# B&R Automation Studio project AGV
Automation Studio 4.12.2.93; technology packages: exosTechnology 2.1.0, mapp 5.20.0, mappCockpit 5.20.0, mappControl 5.20.0, mappMotion 5.20.1, mappView 5.20.0, mappVision 5.20.0

## Configuration CP1586

### Task classes (Cpu.sw)
```
Cyclic#1:
  motorCtrl <- ros_topics_typ.motorCtrl.prg
Binaries: FWRules, TCData, udbdef, User, iomap, Role, arconfig, asfw, ashwac, sysconf, ashwd, target, components
Libraries: ExOS, ExDeploy, ExData, runtime, sys_lib, FileIO, AsIOTime, ArEventLog, AsTCP, ros_topics, ROS, operator, astime, AsIecCon, brsystem, MTTypes, standard
```

## Configuration Config1

CPU X90CP174.48-00, AutomationRuntime B4.91, Build 6.3.0, Safety 0.0, Vc V4.72.6

### Task classes (Cpu.sw)
```
Cyclic#1 (cycle 5000 us, tolerance 0 us):
  motorCtrl <- ros_topics_typ.motorCtrl.prg
  VisionMain <- Package.VisionMain.prg
  WaterTank_ <- (binary)
NcDataObjects: mcdrivelog
Binaries: udbdef, FWRules, TCData, arcoal, arflatprv, arsvcreg, mvLoader, visionUnit, mCoWebSc, iomap, ashwac, Role, sysconf, arconfig, asfw, User, ashwd, target, components, Settings, viApp, viComp, ViLine
Libraries: brsystem, MTTypes, sys_lib, runtime, ROS, standard, ExOS, ExDeploy, ExData, FileIO, AsIOTime, ArEventLog, AsTCP, ros_topics, astime, ViBase, AsZip, AsARCfg, powerlnk, AsEPL, AsIO, MTBasics, MTFilter, AsIecCon, AsIODiag, AsETH, AsBrWStr, AsHttp, AsMem, AsBrStr, CoTrace, McBase, brdkViBase, brdkViCal, brdkViGeom, brdkViImg, brdkViMapp, brdkViVF, brdkWS, MTLinAlg, brdkMU, brdkSTR, AsSem, mpbase, arssl
```

### Hardware
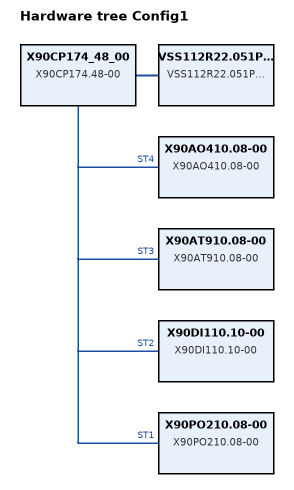
```
VSS112R22.051P-000 : VSS112R22.051P-000 v1.7.0.605  [PLK1 -> X90CP174_48_00.IF3 (NodeNumber=1) [Cable Type=PowerlinkCable, Length=10, Version=1.0.0.3]]
  Supervision = off
  VisionConfig = gCamera
X90AO410.08-00 : X90AO410.08-00 v1.1.0.0  [ST -> X90CP174_48_00.ST4]
X90AT910.08-00 : X90AT910.08-00 v1.0.1.0  [ST -> X90CP174_48_00.ST3]
X90CP174_48_00 : X90CP174.48-00 v1.4.5.0  [X1 -> X1.SL]
  Module X1 (Type=X1, Virtual=true, Version=1.4.5.0)
    Connection (Connector=SL, TargetModule=X90CP174_48_00, TargetConnector=X1)
    ChannelConfig01 = 42
    DigitalFilterPin01 = 0
    ChannelConfig02 = 42
    DigitalFilterPin02 = 0
    ChannelConfig03 = 42
    DigitalFilterPin03 = 0
    ChannelConfig04 = 42
    DigitalFilterPin04 = 0
    IN1_CounterFunction01 = 3
    IN1_CounterFunction02 = 3
    ChannelConfig33 = 15
    PWMSource33 = 1
    PWMSyncPeriod33 = 125
    ChannelConfig34 = 20
    ChannelConfig35 = 20
    ChannelConfig36 = 20  // Configuration and impedance of pin X1.A.J1  
    ChannelConfig37 = 16
    ChannelConfig38 = 20  // Configuration and impedance of pin X1.A.L1  (6A)
    ChannelConfig39 = 20  // Configuration and impedance of pin X1.A.M2 (6A)
    ChannelConfig40 = 20
    ChannelConfig41 = 15
    PWMSource41 = 1
    PWMSyncPeriod41 = 125
    PWMDisplacement41 = 62
    ChannelConfig42 = 20
    ChannelConfig43 = 20  // Configuration and impedance of pin X1.B.H1  (6A)
    ChannelConfig44 = 20  // Configuration and impedance of pin X1.B.H3  (6A)
    ChannelConfig45 = 16  // Configuration and impedance of pin X1.B.G4  (6A)
    ChannelConfig46 = 20
    ChannelConfig47 = 20
    ChannelConfig48 = 20
  Connector IF2:
    ActivateDevice = 1
    Mode = Manual
    InternetAddress = 192.168.87.200
    SubnetMask = 255.255.255.0
    InaNodeNumber = 1
  Connector IF3:
    MtuSize = 1500
    CycleTime = 5000
    InternetAddress = 192.168.200.240
    SubnetMask = 255.255.255.0
  ConfigurationID = AGV_Config1
  UserPartitionSize = 0
  EnableUsbRemoteInstall = 1
  EnableCfRemoteInstall = 1
  TimerDeviceType = EPLX2X
  TimerDevice = X90CP174_48_00.IF3
  TaskClassIdleTime = 5000
  Cyclic1Duration = 5000
  Cyclic1Tolerance = 0
  Cyclic1Stack = 16384
  Cyclic2Duration = 20000
  Cyclic2Tolerance = 20000
  Cyclic3Duration = 50000
  Cyclic3Tolerance = 50000
  Cyclic4Duration = 100000
  Cyclic4Tolerance = 100000
  Cyclic5Duration = 200000
  Cyclic5Tolerance = 200000
  Cyclic6Duration = 500000
  Cyclic6Tolerance = 500000
  Cyclic7Duration = 1000000
  Cyclic7Tolerance = 1000000
  Cyclic8Duration = 10000
  Cyclic8Tolerance = 30000000
  FileDevice1
  FileDeviceName1 = USER
  FileDevicePath1 = USER_PATH
  Route1
  DestinationAddress1 = 10.0.0.2
  SubnetMask1 = 255.255.255.0
  ActivateOpcUa = 1
  OpcUaInformationModels_PV_Version = 2
  OpcUaInformationModel_BaseObjectTypeForStructures = 0
X90DI110.10-00 : X90DI110.10-00 v1.1.1.0  [ST -> X90CP174_48_00.ST2]
X90PO210.08-00 : X90PO210.08-00 v1.4.0.0  [ST -> X90CP174_48_00.ST1]
```

### IoMap.iom - X90CP174_48_00/IoMap.iom
```iecst
VAR_CONFIG
	::motorCtrl:localVariables[0].hw.output.pwm AT %QW."X1".PWMOutput33;
	::motorCtrl:localVariables[0].hw.input.encoder AT %IW."X1".Encoder01;
	::motorCtrl:localVariables[0].hw.input.current[0] AT %IW."X1".Current33;
	::motorCtrl:localVariables[0].hw.input.current[1] AT %IW."X1".Current34;
	::motorCtrl:localVariables[0].hw.input.current[2] AT %IW."X1".Current35;
	::motorCtrl:localVariables[0].hw.input.current[3] AT %IW."X1".Current36;
	::motorCtrl:localVariables[0].hw.input.overload AT %IX."X1".OverloadDigitalOutput33;
	::motorCtrl:localVariables[0].hw.output.clear AT %QX."X1".OverloadClear33;
	::motorCtrl:localVariables[1].hw.input.encoder AT %IW."X1".Encoder02;
	::motorCtrl:localVariables[1].hw.output.pwm AT %QW."X1".PWMOutput37;
	::motorCtrl:localVariables[0].hw.input.current[4] AT %IW."X1".Current37;
	::motorCtrl:localVariables[0].hw.input.current[6] AT %IW."X1".Current39;
	::motorCtrl:localVariables[1].hw.input.nettime AT %ID."X90CP174_48_00".SystemTime;
	::motorCtrl:localVariables[0].hw.input.nettime AT %ID."X90CP174_48_00".SystemTime;
	::motorCtrl:localVariables[0].hw.input.current[5] AT %IW."X1".Current38;
	::motorCtrl:localVariables[0].hw.input.current[7] AT %IW."X1".Current40;
	::motorCtrl:localVariables[1].hw.output.pwm AT %QW."X1".PWMOutput41;
	::motorCtrl:localVariables[1].hw.output.clear AT %QX."X1".OverloadClear41;
	::motorCtrl:localVariables[1].hw.input.current[0] AT %IW."X1".Current41;
	::motorCtrl:localVariables[1].hw.input.overload AT %IX."X1".OverloadDigitalOutput41;
	::motorCtrl:localVariables[1].hw.input.current[1] AT %IW."X1".Current42;
	::motorCtrl:localVariables[1].hw.input.current[2] AT %IW."X1".Current43;
	::motorCtrl:localVariables[1].hw.input.current[3] AT %IW."X1".Current44;
	::motorCtrl:localVariables[1].hw.input.current[4] AT %IW."X1".Current45;
	::motorCtrl:localVariables[1].hw.input.current[5] AT %IW."X1".Current46;
	::motorCtrl:localVariables[1].hw.input.current[6] AT %IW."X1".Current47;
	::motorCtrl:localVariables[1].hw.input.current[7] AT %IW."X1".Current48;
	::VisionMain:hwCam.in.common.moduleOk AT %IX."VSS112R22.051P-000".ModuleOk;
	::VisionMain:hwCam.in.common.serialNumber AT %ID."VSS112R22.051P-000".SerialNumber;
	::VisionMain:hwCam.in.common.moduleId AT %ID."VSS112R22.051P-000".ModuleID;
	::VisionMain:hwCam.in.common.hardwareVariant AT %ID."VSS112R22.051P-000".HardwareVariant;
	::VisionMain:hwCam.in.common.firmwareVersion AT %ID."VSS112R22.051P-000".FirmwareVersion;
	::VisionMain:hwCam.in.status.sensorTemperature AT %IB."VSS112R22.051P-000".SensorTemperature;
	::VisionMain:hwCam.in.status.lightWarningCnt AT %IB."VSS112R22.051P-000".LightWarningCnt;
	::VisionMain:hwCam.out.par.statusLED AT %QB."VSS112R22.051P-000".StatusLED;
	::VisionMain:hwCam.in.status.cameraStatus AT %ID."VSS112R22.051P-000".CameraStatus;
	::VisionMain:hwCam.in.status.acceptedAcquisitionCnt AT %IB."VSS112R22.051P-000".AcceptedAcquisitionCnt;
	::VisionMain:hwCam.in.status.completedAcquisitionCnt AT %IB."VSS112R22.051P-000".CompletedAcquisitionCnt;
	::VisionMain:hwCam.in.status.failedAcquisitionCnt AT %IB."VSS112R22.051P-000".FailedAcquisitionCnt;
	::VisionMain:hwCam.in.status.gainLevel AT %IB."VSS112R22.051P-000".ReadGainLevel;
	::VisionMain:hwCam.in.status.focus AT %IW."VSS112R22.051P-000".ReadFocus;
	::VisionMain:hwCam.in.status.exposureTime AT %ID."VSS112R22.051P-000".ReadExposureTime;
	::VisionMain:hwCam.out.par.gainLevel AT %QB."VSS112R22.051P-000".GainLevel;
	::VisionMain:hwCam.out.par.focus AT %QW."VSS112R22.051P-000".SetFocus;
	::VisionMain:hwCam.out.par.exposureTime AT %QD."VSS112R22.051P-000".ExposureTime01;
	::VisionMain:hwCam.out.par.delayNetTime AT %QD."VSS112R22.051P-000".DelayNettime01;
	::VisionMain:hwCam.out.par.flashColor AT %QB."VSS112R22.051P-000".FlashColor01;
	::VisionMain:hwCam.out.par.flashSegment AT %QB."VSS112R22.051P-000".FlashSegment01;
	::VisionMain:hwCam.in.status.undervoltageError AT %IX."VSS112R22.051P-000".UndervoltageError;
	::VisionMain:hwCam.in.status.digitalInput AT %IX."VSS112R22.051P-000".DigitalInput01;
	::VisionMain:hwCam.out.cmd.digitalOutput AT %QX."VSS112R22.051P-000".DigitalOutput01;
	::VisionMain:hwCam.in.status.digitalOutputStatus AT %IX."VSS112R22.051P-000".DigitalOutputStatus01;
	::VisionMain:hwCam.in.status.imageAcquisitionReady AT %IX."VSS112R22.051P-000".ImageAcquisitionReady;
	::VisionMain:hwCam.in.status.imageProcessingActive AT %IX."VSS112R22.051P-000".ImageProcessingActive;
	::VisionMain:hwCam.out.cmd.imageAcquisition AT %QX."VSS112R22.051P-000".ImageAcquisition;
	::VisionMain:hwCam.out.cmd.resetAcquisiton AT %QX."VSS112R22.051P-000".ResetAcquisition;
	::VisionMain:hwCam.out.cmd.searchAcquisitonSettings AT %QX."VSS112R22.051P-000".SearchAcquisitionSettings;
	::VisionMain:hwCam.out.par.IRFilter AT %QX."VSS112R22.051P-000".IRFilter;
	::VisionMain:hwCam.out.par.chromaticLock AT %QX."VSS112R22.051P-000".ChromaticLock;
	::VisionMain:hwCam.in.status.cameraProcessingTime AT %IW."VSS112R22.051P-000".CameraProcessingTime;
	::VisionMain:hwCam.in.status.imageProcessingError AT %IW."VSS112R22.051P-000".ImageProcessingError;
	::VisionMain:hwCam.in.status.imageNettime AT %ID."VSS112R22.051P-000".ImageNettime;
	::VisionMain:hwBlob.out.common.enable AT %QX."VSS112R22.051P-000".Enable;
	::VisionMain:hwBlob.out.common.numSearchMax AT %QB."VSS112R22.051P-000".NumSearchMax;
	::VisionMain:hwBlob.out.regionFeatures AT %QX."VSS112R22.051P-000".RegionalFeatures;
	::VisionMain:hwBlob.out.enhancedBlobInformation AT %QX."VSS112R22.051P-000".EnhancedBlobInfo;
	::VisionMain:hwBlob.out.common.alignment AT %QB."VSS112R22.051P-000".Alignment;
	::VisionMain:hwBlob.out.common.offsetROI.x AT %QD."VSS112R22.051P-000".OffsetRoiX;
	::VisionMain:hwBlob.out.common.offsetROI.y AT %QD."VSS112R22.051P-000".OffsetRoiY;
	::VisionMain:hwBlob.out.common.offsetROI.orientation AT %QW."VSS112R22.051P-000".OffsetRoiOrientation;
	::VisionMain:hwBlob.out.common.offsetROI.rotCenterX AT %QD."VSS112R22.051P-000".OffsetRoiRotationCenterX;
	::VisionMain:hwBlob.out.common.offsetROI.rotCenterY AT %QD."VSS112R22.051P-000".OffsetRoiRotationCenterY;
	::VisionMain:hwBlob.in.results[0].xMin AT %ID."VSS112R22.051P-000".BlobXMin01;
	::VisionMain:hwBlob.in.results[0].xMax AT %ID."VSS112R22.051P-000".BlobXMax01;
	::VisionMain:hwBlob.in.results[0].yMin AT %ID."VSS112R22.051P-000".BlobYMin01;
	::VisionMain:hwBlob.in.results[0].yMax AT %ID."VSS112R22.051P-000".BlobYMax01;
	::VisionMain:hwBlob.in.common.numResults AT %IB."VSS112R22.051P-000".NumRes;
	::motorCtrl:suction.valveEnable AT %QX."X90PO210.08-00".DigitalOutput01;
	::motorCtrl:suction.motorEnable AT %QX."X90PO210.08-00".DigitalOutput02;
	::VisionMain:hwBlob.in.results[0].area AT %ID."VSS112R22.051P-000".blobArea01;
	::VisionMain:hwBlob.in.results[1].area AT %ID."VSS112R22.051P-000".blobArea02;
	::VisionMain:hwBlob.in.results[1].xMin AT %ID."VSS112R22.051P-000".BlobXMin02;
	::VisionMain:hwBlob.in.results[1].xMax AT %ID."VSS112R22.051P-000".BlobXMax02;
	::VisionMain:hwBlob.in.results[1].yMin AT %ID."VSS112R22.051P-000".BlobYMin02;
	::VisionMain:hwBlob.in.results[1].yMax AT %ID."VSS112R22.051P-000".BlobYMax02;
	::VisionMain:hwBlob.in.results[0].modelNumber AT %IB."VSS112R22.051P-000".model01;
	::VisionMain:hwBlob.in.results[1].modelNumber AT %IB."VSS112R22.051P-000".model02;
	::VisionMain:hwBlob.in.results[2].modelNumber AT %IB."VSS112R22.051P-000".model03;
	::VisionMain:hwBlob.in.results[3].modelNumber AT %IB."VSS112R22.051P-000".model04;
	::VisionMain:hwBlob.in.results[2].area AT %ID."VSS112R22.051P-000".blobArea03;
	::VisionMain:hwBlob.in.results[3].area AT %ID."VSS112R22.051P-000".blobArea04;
	::VisionMain:hwBlob.in.results[2].xMin AT %ID."VSS112R22.051P-000".BlobXMin03;
	::VisionMain:hwBlob.in.results[3].xMin AT %ID."VSS112R22.051P-000".BlobXMin04;
	::VisionMain:hwBlob.in.results[2].xMax AT %ID."VSS112R22.051P-000".BlobXMax03;
	::VisionMain:hwBlob.in.results[3].xMax AT %ID."VSS112R22.051P-000".BlobXMax04;
	::VisionMain:hwBlob.in.results[2].yMin AT %ID."VSS112R22.051P-000".BlobYMin03;
	::VisionMain:hwBlob.in.results[3].yMin AT %ID."VSS112R22.051P-000".BlobYMin04;
	::VisionMain:hwBlob.in.results[2].yMax AT %ID."VSS112R22.051P-000".BlobYMax03;
	::VisionMain:hwBlob.in.results[3].yMax AT %ID."VSS112R22.051P-000".BlobYMax04;
	::VisionMain:hwBlob.in.results[0].positionX AT %ID."VSS112R22.051P-000".posX01;
	::VisionMain:hwBlob.in.results[1].positionX AT %ID."VSS112R22.051P-000".posX02;
	::VisionMain:hwBlob.in.results[2].positionX AT %ID."VSS112R22.051P-000".posX03;
	::VisionMain:hwBlob.in.results[3].positionX AT %ID."VSS112R22.051P-000".posX04;
	::VisionMain:hwBlob.in.results[0].positionY AT %ID."VSS112R22.051P-000".posY01;
	::VisionMain:hwBlob.in.results[1].positionY AT %ID."VSS112R22.051P-000".posY02;
	::VisionMain:hwBlob.in.results[2].positionY AT %ID."VSS112R22.051P-000".posY03;
	::VisionMain:hwBlob.in.results[3].positionY AT %ID."VSS112R22.051P-000".posY04;
	::VisionMain:hwBlob.in.results[0].circularity AT %IB."VSS112R22.051P-000".blobCirc01;
	::VisionMain:hwBlob.in.results[1].circularity AT %IB."VSS112R22.051P-000".blobCirc02;
	::VisionMain:hwBlob.in.results[2].circularity AT %IB."VSS112R22.051P-000".blobCirc03;
	::VisionMain:hwBlob.in.results[3].circularity AT %IB."VSS112R22.051P-000".blobCirc04;
	::VisionMain:hwBlob.in.results[0].rectangularity AT %IB."VSS112R22.051P-000".blobRect01;
	::VisionMain:hwBlob.in.results[1].rectangularity  AT %IB."VSS112R22.051P-000".blobRect02;
	::VisionMain:hwBlob.in.results[2].rectangularity  AT %IB."VSS112R22.051P-000".blobRect03;
	::VisionMain:hwBlob.in.results[3].rectangularity  AT %IB."VSS112R22.051P-000".blobRect04;
END_VAR
```

### target.exostarget - X90CP174_48_00/exosTechnology/target.exostarget
```
Element gTarget_0 (Type=exostarget)
  General:
    ConnectionIP = 192.168.87.42
    Logging:
      LogLevel = Success
      LogFilters:
        LogFilterUser = On
        LogFilterSystem = On
        LogFilterVerbose = Off
      LogDestination = Volatile
    Deployment = On
      MaxRestarts = 10
    DataConnection = On
      ConnectionType = TCPIP
      TimeSynchronization:
        TimeConnection:
          TimePort = 49001
        PrecisionUsec = 5000
        GuardTimeSec = 180
        DeviationPerHourUsec = 100000
      DataConnectionLogging:
        LogConnection:
          LogPort = 49002
          LogShmPath = exos_log
        LogCycleTimeMsec = 50
  Components:
    ComponentsGeneral:
      ComponentsHeartbeatMsec = 500
      ComponentsTimeoutSec = 2
      ComponentsTaskClass = 2
      ComponentsCycleTimeMsec = 10
    Component[0]:
      ComponentConfigurationLink = gros_topics_typ_0
      DataModels:
        Instance[0]:
          InstanceName = ros_topics_typ_0
          InstanceConnection:
            InstancePort = 49005
            InstanceShmPath = ros_topics_typ_0
  ComponentDataConnection:
    Version = 2.1.0-1
    ErrorHandling = Target
    RestartEvent = Target
    StartupTimeout = 5
    Predefined:
      Files:
        File[0]:
          FileName = ufw-exos-data
          ChangeEvent = Ignore
        File[1]:
          FileName = exos-data-ufw-profile.sh
          ChangeEvent = Ignore
        File[2]:
          FileName = exos-data-ports-allow.sh
          ChangeEvent = Restart
        File[3]:
          FileName = exos-data.conf
          ChangeEvent = Restart
        File[4]:
          FileName = exos-data_2.1.0-1_amd64.deb
          ChangeEvent = Reinstall
        File[5]:
          FileName = exos-data-eth_2.1.0-1_amd64.deb
          ChangeEvent = Reinstall
        File[6]:
          FileName = exos-data-remove.sh
          ChangeEvent = Ignore
        File[7]:
          FileName = run_server.sh
          ChangeEvent = Ignore
        File[8]:
          FileName = setup_build_environment.sh
          ChangeEvent = Ignore
        File[9]:
          FileName = libzmq5_4.2.1-4+deb9u2_amd64.deb
          ChangeEvent = Reinstall
        File[10]:
          FileName = libpgm-5.2-0_5.2.122~dfsg-2_amd64.deb
          ChangeEvent = Reinstall
        File[11]:
          FileName = libsodium18_1.0.11-2_amd64.deb
          ChangeEvent = Reinstall
      Services:
        Service[0]:
          Type = Install
          Command = dpkg -i *.deb
          WorkingDirectory
        Service[1]:
          Type = Remove
          Command = dpkg --purge exos-data
          WorkingDirectory
        Service[2]:
          Type = Remove
          Command = dpkg --purge exos-data-eth
          WorkingDirectory
        Service[3]:
          Type = Remove
          Command = sh exos-data-remove.sh
          WorkingDirectory
        Service[4]:
          Type = Startup
          Command = cp exos-data.conf /etc/exos-data.conf
          WorkingDirectory
        Service[5]:
          Type = Startup
          Command = sh exos-data-ufw-profile.sh
          WorkingDirectory
        Service[6]:
          Type = Startup
          Command = sh exos-data-ports-allow.sh
          WorkingDirectory
        Service[7]:
          Type = Runtime
          Command = /usr/bin/exos_mr
          WorkingDirectory
  Simulation:
    SimConnectionIP = 192.168.87.42
    SimDeployment = On
    SimDataConnection = On
      SimConnectionType = TCPIP
      SimTimeSynchronization:
        SimPrecisionUsec = 10000
        SimGuardTimeSec = 30
    SimComponentsGeneral:
      SimComponentsHeartbeatMsec = 1000
      SimComponentsTimeoutSec = 75
```

### viComp.visioncomponent - X90CP174_48_00/mappVision/viComp.visioncomponent
```
Element gCamera (Type=visioncomponent)
  VisionApplicationReference = ViLine
```

## Logical view

Binary libraries used (declarations not repeated): operator, runtime, astime, AsIecCon, brsystem, standard, MTTypes, sys_lib, ROS, FileIO, AsIOTime, ArEventLog, AsTCP, ExOS, ExDeploy, ExData, AsZip, AsARCfg, powerlnk, AsEPL, AsIO, AsIODiag, AsETH, AsBrWStr, AsHttp, AsMem, AsBrStr, brdkViBase 1.00.4, brdkViCal, brdkViGeom, brdkViImg, brdkViMapp, brdkViVF, brdkWS, McBase 5.20.1, ViBase, CoTrace, MTBasics 5.20.0, MTFilter 5.20.0, MTLinAlg, brdkMU, brdkSTR, AsSem

### Global.var - Global variables
```iecst
VAR
	updateLineStatus : BOOL;
	sharpTurn : BOOL;
	rightTurn : BOOL;
	orientationReached : BOOL := TRUE;
	lineMode : BOOL;
	drejMere : REAL;
	Test2 : INT;
	slowDown : REAL;
	angVel : LREAL;
	holdRight : BOOL;
	lineFollow : ros_lineMode;
	moveForward : BOOL;
	lineStatus : ros_lineStatus;
	awaitDecision : BOOL;
	tempDec : BOOL;
	sammenEnable : BOOL;
END_VAR
```

### Package Logical/Libraries - Global libraries

- ros_topics_typ.exospkg (not shown)

### exos_ros_topics_typ.h - Generated datamodel header for ros_topics_typ
```c
/*Automatically generated header file from ros_topics_typ.typ*/

#ifndef _EXOS_COMP_ROS_TOPICS_TYP_H_
#define _EXOS_COMP_ROS_TOPICS_TYP_H_

#include "exos_api.h"

#if defined(_SG4)
#include <ros_topics.h>
#else
#include <stddef.h>
#include <stdint.h>
#include <stdbool.h>

typedef struct ros_lineStatus
{
    int16_t lineStatusCode;

} ros_lineStatus;

typedef struct ros_lineMode
{
    bool lineMode;
    bool lineSharpTurn;
    bool lineHoldRight;
    bool lineForward;
    bool lineInterSection;
    bool lineDecision;
    bool lineFast;
    bool lineSlow;

} ros_lineMode;

typedef struct ros_armBools
{
    bool vaccumValve;
    bool vaccumMotor;

} ros_armBools;

typedef struct ros_encoder
{
    int16_t encoder1;
    int16_t encoder2;

} ros_encoder;

typedef struct ros_config_typ
{
    double maxSpeed;
    double minSpeed;
    double baseWidth;

} ros_config_typ;

typedef struct ros_topic_vector3_typ
{
    double y;
    double z;
    double x;

} ros_topic_vector3_typ;

typedef struct ros_topic_twist_typ
{
    struct ros_topic_vector3_typ angular;
    struct ros_topic_vector3_typ linear;

} ros_topic_twist_typ;

typedef struct ros_topic_time_typ
{
    uint32_t nsec;
    uint32_t sec;

} ros_topic_time_typ;

typedef struct ros_topic_header_typ
{
    struct ros_topic_time_typ stamp;
    uint32_t seq;
    char frame_id[21];

} ros_topic_header_typ;

typedef struct ros_topic_twistCor_typ
{
    struct ros_topic_twist_typ twist;

} ros_topic_twistCor_typ;

typedef struct ros_topic_quaternion_typ
{
    double y;
    double z;
    double w;
    double x;

} ros_topic_quaternion_typ;

typedef struct ros_topic_point_typ
{
    double y;
    double z;
    double x;

} ros_topic_point_typ;

typedef struct ros_topic_pose_typ
{
    struct ros_topic_point_typ position;
    struct ros_topic_quaternion_typ orientation;

} ros_topic_pose_typ;

typedef struct ros_topic_poseCor_typ
{
    struct ros_topic_pose_typ pose;

} ros_topic_poseCor_typ;

typedef struct ros_topic_odemety_typ
{
    struct ros_topic_poseCor_typ pose;
    struct ros_topic_twistCor_typ twist;
    struct ros_topic_header_typ header;

} ros_topic_odemety_typ;

typedef struct ros_topics_typ
{
    struct ros_topic_odemety_typ odemetry; //PUB
    struct ros_topic_twist_typ twist; //SUB
    struct ros_config_typ config; //SUB
    struct ros_encoder encoder; //PUB
    struct ros_armBools vaccumTopic; //SUB
    struct ros_lineMode lineFollow; //SUB
    struct ros_lineStatus lineStatus; //PUB

} ros_topics_typ;

#endif // _SG4

EXOS_ERROR_CODE exos_datamodel_connect_ros_topics_typ(exos_datamodel_handle_t *datamodel, exos_datamodel_event_cb datamodel_event_callback);

#endif // _EXOS_COMP_ROS_TOPICS_TYP_H_
```

### libros_topics_typ.h - ros_topics_typ static library wrapper header
```c
#ifndef _LIBROS_TOPICS_TYP_H_
#define _LIBROS_TOPICS_TYP_H_

#include "exos_ros_topics_typ.h"

typedef void (*libros_topics_typ_event_cb)(void);
typedef void (*libros_topics_typ_method_fn)(void);
typedef int32_t (*libros_topics_typ_get_nettime_fn)(void);
typedef void (*libros_topics_typ_log_fn)(char *log_entry);

typedef struct libros_topics_typodemetry
{
    libros_topics_typ_event_cb on_change;
    int32_t nettime;
    ros_topic_odemety_typ value;
} libros_topics_typodemetry_t;

typedef struct libros_topics_typtwist
{
    libros_topics_typ_method_fn publish;
    ros_topic_twist_typ value;
} libros_topics_typtwist_t;

typedef struct libros_topics_typconfig
{
    libros_topics_typ_method_fn publish;
    ros_config_typ value;
} libros_topics_typconfig_t;

typedef struct libros_topics_typencoder
{
    libros_topics_typ_event_cb on_change;
    int32_t nettime;
    ros_encoder value;
} libros_topics_typencoder_t;

typedef struct libros_topics_typvaccumTopic
{
    libros_topics_typ_method_fn publish;
    ros_armBools value;
} libros_topics_typvaccumTopic_t;

typedef struct libros_topics_typlineFollow
{
    libros_topics_typ_method_fn publish;
    ros_lineMode value;
} libros_topics_typlineFollow_t;

typedef struct libros_topics_typlineStatus
{
    libros_topics_typ_event_cb on_change;
    int32_t nettime;
    ros_lineStatus value;
} libros_topics_typlineStatus_t;

typedef struct libros_topics_typ_log
{
    libros_topics_typ_log_fn error;
    libros_topics_typ_log_fn warning;
    libros_topics_typ_log_fn success;
    libros_topics_typ_log_fn info;
    libros_topics_typ_log_fn debug;
    libros_topics_typ_log_fn verbose;
} libros_topics_typ_log_t;

typedef struct libros_topics_typ
{
    libros_topics_typ_method_fn connect;
    libros_topics_typ_method_fn disconnect;
    libros_topics_typ_method_fn process;
    libros_topics_typ_method_fn set_operational;
    libros_topics_typ_method_fn dispose;
    libros_topics_typ_get_nettime_fn get_nettime;
    libros_topics_typ_log_t log;
    libros_topics_typ_event_cb on_connected;
    libros_topics_typ_event_cb on_disconnected;
    libros_topics_typ_event_cb on_operational;
    bool is_connected;
    bool is_operational;
    libros_topics_typodemetry_t odemetry;
    libros_topics_typtwist_t twist;
    libros_topics_typconfig_t config;
    libros_topics_typencoder_t encoder;
    libros_topics_typvaccumTopic_t vaccumTopic;
    libros_topics_typlineFollow_t lineFollow;
    libros_topics_typlineStatus_t lineStatus;
} libros_topics_typ_t;

#ifdef __cplusplus
extern "C" {
#endif
libros_topics_typ_t *libros_topics_typ_init(void);
#ifdef __cplusplus
}
#endif
#endif // _LIBROS_TOPICS_TYP_H_
```

### libros_topics_typ.c - ros_topics_typ static library wrapper source
```c
#include <string.h>
#define EXOS_ASSERT_LOG &logger
#include "exos_log.h"
#include "libros_topics_typ.h"

#define SUCCESS(_format_, ...) exos_log_success(&logger, EXOS_LOG_TYPE_USER, _format_, ##__VA_ARGS__);
#define INFO(_format_, ...) exos_log_info(&logger, EXOS_LOG_TYPE_USER, _format_, ##__VA_ARGS__);
#define VERBOSE(_format_, ...) exos_log_debug(&logger, EXOS_LOG_TYPE_USER + EXOS_LOG_TYPE_VERBOSE, _format_, ##__VA_ARGS__);
#define ERROR(_format_, ...) exos_log_error(&logger, _format_, ##__VA_ARGS__);

static exos_log_handle_t logger;

typedef struct libros_topics_typHandle
{
    libros_topics_typ_t ext_ros_topics_typ_datamodel;
    exos_datamodel_handle_t ros_topics_typ_datamodel;

    exos_dataset_handle_t odemetry_dataset;
    exos_dataset_handle_t twist_dataset;
    exos_dataset_handle_t config_dataset;
    exos_dataset_handle_t encoder_dataset;
    exos_dataset_handle_t vaccumtopic;
    exos_dataset_handle_t linefollow;
    exos_dataset_handle_t linestatus;
} libros_topics_typHandle_t;

static libros_topics_typHandle_t h_ros_topics_typ;

static void libros_topics_typ_datasetEvent(exos_dataset_handle_t *dataset, EXOS_DATASET_EVENT_TYPE event_type, void *info)
{
    switch (event_type)
    {
    case EXOS_DATASET_EVENT_UPDATED:
        VERBOSE("dataset %s updated! latency (us):%i", dataset->name, (exos_datamodel_get_nettime(dataset->datamodel) - dataset->nettime));
        //handle each subscription dataset separately
        if (0 == strcmp(dataset->name, "odemetry"))
        {
            //update the nettime
            h_ros_topics_typ.ext_ros_topics_typ_datamodel.odemetry.nettime = dataset->nettime;

            //trigger the callback if assigned
            if (NULL != h_ros_topics_typ.ext_ros_topics_typ_datamodel.odemetry.on_change)
            {
                h_ros_topics_typ.ext_ros_topics_typ_datamodel.odemetry.on_change();
            }
        }
        else if (0 == strcmp(dataset->name, "encoder"))
        {
            //update the nettime
            h_ros_topics_typ.ext_ros_topics_typ_datamodel.encoder.nettime = dataset->nettime;

            //trigger the callback if assigned
            if (NULL != h_ros_topics_typ.ext_ros_topics_typ_datamodel.encoder.on_change)
            {
                h_ros_topics_typ.ext_ros_topics_typ_datamodel.encoder.on_change();
            }
        }
        else if (0 == strcmp(dataset->name, "lineStatus"))
        {
            //update the nettime
            h_ros_topics_typ.ext_ros_topics_typ_datamodel.lineStatus.nettime = dataset->nettime;

            //trigger the callback if assigned
            if (NULL != h_ros_topics_typ.ext_ros_topics_typ_datamodel.lineStatus.on_change)
            {
                h_ros_topics_typ.ext_ros_topics_typ_datamodel.lineStatus.on_change();
            }
        }
        break;

    case EXOS_DATASET_EVENT_PUBLISHED:
        break;
    case EXOS_DATASET_EVENT_DELIVERED:
        break;
    case EXOS_DATASET_EVENT_CONNECTION_CHANGED:
        INFO("dataset %s changed state to %s", dataset->name, exos_get_state_string(dataset->connection_state));

        switch (dataset->connection_state)
        {
        case EXOS_STATE_DISCONNECTED:
            break;
        case EXOS_STATE_CONNECTED:
            break;
        case EXOS_STATE_OPERATIONAL:
            break;
        case EXOS_STATE_ABORTED:
            ERROR("dataset %s error %d (%s) occured", dataset->name, dataset->error, exos_get_error_string(dataset->error));
            break;
        }
        break;
    }
}

static void libros_topics_typ_datamodelEvent(exos_datamodel_handle_t *datamodel, const EXOS_DATAMODEL_EVENT_TYPE event_type, void *info)
{
    switch (event_type)
    {
    case EXOS_DATAMODEL_EVENT_CONNECTION_CHANGED:
        INFO("application changed state to %s", exos_get_state_string(datamodel->connection_state));

        h_ros_topics_typ.ext_ros_topics_typ_datamodel.is_connected = false;
        h_ros_topics_typ.ext_ros_topics_typ_datamodel.is_operational = false;
        switch (datamodel->connection_state)
        {
        case EXOS_STATE_DISCONNECTED:
            if (NULL != h_ros_topics_typ.ext_ros_topics_typ_datamodel.on_disconnected)
            {
                h_ros_topics_typ.ext_ros_topics_typ_datamodel.on_disconnected();
            }
            break;
        case EXOS_STATE_CONNECTED:
            h_ros_topics_typ.ext_ros_topics_typ_datamodel.is_connected = true;
            if (NULL != h_ros_topics_typ.ext_ros_topics_typ_datamodel.on_connected)
            {
                h_ros_topics_typ.ext_ros_topics_typ_datamodel.on_connected();
            }
            break;
        case EXOS_STATE_OPERATIONAL:
            h_ros_topics_typ.ext_ros_topics_typ_datamodel.is_connected = true;
            h_ros_topics_typ.ext_ros_topics_typ_datamodel.is_operational = true;
            if (NULL != h_ros_topics_typ.ext_ros_topics_typ_datamodel.on_operational)
            {
                h_ros_topics_typ.ext_ros_topics_typ_datamodel.on_operational();
            }
            SUCCESS("ros_topics_typ operational!");
            break;
        case EXOS_STATE_ABORTED:
            if (NULL != h_ros_topics_typ.ext_ros_topics_typ_datamodel.on_disconnected)
            {
                h_ros_topics_typ.ext_ros_topics_typ_datamodel.on_disconnected();
            }
            ERROR("application error %d (%s) occured", datamodel->error, exos_get_error_string(datamodel->error));
            break;
        }
        break;
    case EXOS_DATAMODEL_EVENT_SYNC_STATE_CHANGED:
        break;

    default:
        break;

    }
}

static void libros_topics_typ_publish_twist_dataset(void)
{
    EXOS_ASSERT_OK(exos_dataset_publish(&h_ros_topics_typ.twist_dataset));
}
static void libros_topics_typ_publish_config_dataset(void)
{
    EXOS_ASSERT_OK(exos_dataset_publish(&h_ros_topics_typ.config_dataset));
}
static void libros_topics_typ_publish_vaccumtopic(void)
{
    EXOS_ASSERT_OK(exos_dataset_publish(&h_ros_topics_typ.vaccumtopic));
}
static void libros_topics_typ_publish_linefollow(void)
{
    EXOS_ASSERT_OK(exos_dataset_publish(&h_ros_topics_typ.linefollow));
}

static void libros_topics_typ_connect(void)
{
    //connect the datamodel
    EXOS_ASSERT_OK(exos_datamodel_connect_ros_topics_typ(&(h_ros_topics_typ.ros_topics_typ_datamodel), libros_topics_typ_datamodelEvent));

    //connect datasets
    EXOS_ASSERT_OK(exos_dataset_connect(&(h_ros_topics_typ.odemetry_dataset), EXOS_DATASET_SUBSCRIBE, libros_topics_typ_datasetEvent));
    EXOS_ASSERT_OK(exos_dataset_connect(&(h_ros_topics_typ.twist_dataset), EXOS_DATASET_PUBLISH, libros_topics_typ_datasetEvent));
    EXOS_ASSERT_OK(exos_dataset_connect(&(h_ros_topics_typ.config_dataset), EXOS_DATASET_PUBLISH, libros_topics_typ_datasetEvent));
    EXOS_ASSERT_OK(exos_dataset_connect(&(h_ros_topics_typ.encoder_dataset), EXOS_DATASET_SUBSCRIBE, libros_topics_typ_datasetEvent));
    EXOS_ASSERT_OK(exos_dataset_connect(&(h_ros_topics_typ.vaccumtopic), EXOS_DATASET_PUBLISH, libros_topics_typ_datasetEvent));
    EXOS_ASSERT_OK(exos_dataset_connect(&(h_ros_topics_typ.linefollow), EXOS_DATASET_PUBLISH, libros_topics_typ_datasetEvent));
    EXOS_ASSERT_OK(exos_dataset_connect(&(h_ros_topics_typ.linestatus), EXOS_DATASET_SUBSCRIBE, libros_topics_typ_datasetEvent));
}
static void libros_topics_typ_disconnect(void)
{
    h_ros_topics_typ.ext_ros_topics_typ_datamodel.is_connected = false;
    h_ros_topics_typ.ext_ros_topics_typ_datamodel.is_operational = false;

    EXOS_ASSERT_OK(exos_datamodel_disconnect(&(h_ros_topics_typ.ros_topics_typ_datamodel)));
}

static void libros_topics_typ_set_operational(void)
{
    EXOS_ASSERT_OK(exos_datamodel_set_operational(&(h_ros_topics_typ.ros_topics_typ_datamodel)));
}

static void libros_topics_typ_process(void)
{
    EXOS_ASSERT_OK(exos_datamodel_process(&(h_ros_topics_typ.ros_topics_typ_datamodel)));
    exos_log_process(&logger);
}

static void libros_topics_typ_dispose(void)
{
    h_ros_topics_typ.ext_ros_topics_typ_datamodel.is_connected = false;
    h_ros_topics_typ.ext_ros_topics_typ_datamodel.is_operational = false;

    EXOS_ASSERT_OK(exos_datamodel_delete(&(h_ros_topics_typ.ros_topics_typ_datamodel)));
    exos_log_delete(&logger);
}

static int32_t libros_topics_typ_get_nettime(void)
{
    return exos_datamodel_get_nettime(&(h_ros_topics_typ.ros_topics_typ_datamodel));
}

static void libros_topics_typ_log_error(char* log_entry)
{
    exos_log_error(&logger, log_entry);
}

static void libros_topics_typ_log_warning(char* log_entry)
{
    exos_log_warning(&logger, EXOS_LOG_TYPE_USER, log_entry);
}

static void libros_topics_typ_log_success(char* log_entry)
{
    exos_log_success(&logger, EXOS_LOG_TYPE_USER, log_entry);
}

static void libros_topics_typ_log_info(char* log_entry)
{
    exos_log_info(&logger, EXOS_LOG_TYPE_USER, log_entry);
}

static void libros_topics_typ_log_debug(char* log_entry)
{
    exos_log_debug(&logger, EXOS_LOG_TYPE_USER, log_entry);
}

static void libros_topics_typ_log_verbose(char* log_entry)
{
    exos_log_warning(&logger, EXOS_LOG_TYPE_USER + EXOS_LOG_TYPE_VERBOSE, log_entry);
}

libros_topics_typ_t *libros_topics_typ_init(void)
{
    memset(&h_ros_topics_typ, 0, sizeof(h_ros_topics_typ));

    h_ros_topics_typ.ext_ros_topics_typ_datamodel.twist.publish = libros_topics_typ_publish_twist_dataset;
    h_ros_topics_typ.ext_ros_topics_typ_datamodel.config.publish = libros_topics_typ_publish_config_dataset;
    h_ros_topics_typ.ext_ros_topics_typ_datamodel.vaccumTopic.publish = libros_topics_typ_publish_vaccumtopic;
    h_ros_topics_typ.ext_ros_topics_typ_datamodel.lineFollow.publish = libros_topics_typ_publish_linefollow;

    h_ros_topics_typ.ext_ros_topics_typ_datamodel.connect = libros_topics_typ_connect;
    h_ros_topics_typ.ext_ros_topics_typ_datamodel.disconnect = libros_topics_typ_disconnect;
    h_ros_topics_typ.ext_ros_topics_typ_datamodel.process = libros_topics_typ_process;
    h_ros_topics_typ.ext_ros_topics_typ_datamodel.set_operational = libros_topics_typ_set_operational;
    h_ros_topics_typ.ext_ros_topics_typ_datamodel.dispose = libros_topics_typ_dispose;
    h_ros_topics_typ.ext_ros_topics_typ_datamodel.get_nettime = libros_topics_typ_get_nettime;
    h_ros_topics_typ.ext_ros_topics_typ_datamodel.log.error = libros_topics_typ_log_error;
    h_ros_topics_typ.ext_ros_topics_typ_datamodel.log.warning = libros_topics_typ_log_warning;
    h_ros_topics_typ.ext_ros_topics_typ_datamodel.log.success = libros_topics_typ_log_success;
    h_ros_topics_typ.ext_ros_topics_typ_datamodel.log.info = libros_topics_typ_log_info;
    h_ros_topics_typ.ext_ros_topics_typ_datamodel.log.debug = libros_topics_typ_log_debug;
    h_ros_topics_typ.ext_ros_topics_typ_datamodel.log.verbose = libros_topics_typ_log_verbose;

    exos_log_init(&logger, "gros_topics_typ_0");

    SUCCESS("starting gros_topics_typ_0 application..");

    EXOS_ASSERT_OK(exos_datamodel_init(&h_ros_topics_typ.ros_topics_typ_datamodel, "ros_topics_typ_0", "gros_topics_typ_0"));

    //set the user_context to access custom data in the callbacks
    h_ros_topics_typ.ros_topics_typ_datamodel.user_context = NULL; //not used
    h_ros_topics_typ.ros_topics_typ_datamodel.user_tag = 0; //not used

    EXOS_ASSERT_OK(exos_dataset_init(&h_ros_topics_typ.odemetry_dataset, &h_ros_topics_typ.ros_topics_typ_datamodel, "odemetry", &h_ros_topics_typ.ext_ros_topics_typ_datamodel.odemetry.value, sizeof(h_ros_topics_typ.ext_ros_topics_typ_datamodel.odemetry.value)));
    h_ros_topics_typ.odemetry_dataset.user_context = NULL; //not used
    h_ros_topics_typ.odemetry_dataset.user_tag = 0; //not used

    EXOS_ASSERT_OK(exos_dataset_init(&h_ros_topics_typ.twist_dataset, &h_ros_topics_typ.ros_topics_typ_datamodel, "twist", &h_ros_topics_typ.ext_ros_topics_typ_datamodel.twist.value, sizeof(h_ros_topics_typ.ext_ros_topics_typ_datamodel.twist.value)));
    h_ros_topics_typ.twist_dataset.user_context = NULL; //not used
    h_ros_topics_typ.twist_dataset.user_tag = 0; //not used

    EXOS_ASSERT_OK(exos_dataset_init(&h_ros_topics_typ.config_dataset, &h_ros_topics_typ.ros_topics_typ_datamodel, "config", &h_ros_topics_typ.ext_ros_topics_typ_datamodel.config.value, sizeof(h_ros_topics_typ.ext_ros_topics_typ_datamodel.config.value)));
    h_ros_topics_typ.config_dataset.user_context = NULL; //not used
    h_ros_topics_typ.config_dataset.user_tag = 0; //not used

    EXOS_ASSERT_OK(exos_dataset_init(&h_ros_topics_typ.encoder_dataset, &h_ros_topics_typ.ros_topics_typ_datamodel, "encoder", &h_ros_topics_typ.ext_ros_topics_typ_datamodel.encoder.value, sizeof(h_ros_topics_typ.ext_ros_topics_typ_datamodel.encoder.value)));
    h_ros_topics_typ.encoder_dataset.user_context = NULL; //not used
    h_ros_topics_typ.encoder_dataset.user_tag = 0; //not used

    EXOS_ASSERT_OK(exos_dataset_init(&h_ros_topics_typ.vaccumtopic, &h_ros_topics_typ.ros_topics_typ_datamodel, "vaccumTopic", &h_ros_topics_typ.ext_ros_topics_typ_datamodel.vaccumTopic.value, sizeof(h_ros_topics_typ.ext_ros_topics_typ_datamodel.vaccumTopic.value)));
    h_ros_topics_typ.vaccumtopic.user_context = NULL; //not used
    h_ros_topics_typ.vaccumtopic.user_tag = 0; //not used

    EXOS_ASSERT_OK(exos_dataset_init(&h_ros_topics_typ.linefollow, &h_ros_topics_typ.ros_topics_typ_datamodel, "lineFollow", &h_ros_topics_typ.ext_ros_topics_typ_datamodel.lineFollow.value, sizeof(h_ros_topics_typ.ext_ros_topics_typ_datamodel.lineFollow.value)));
    h_ros_topics_typ.linefollow.user_context = NULL; //not used
    h_ros_topics_typ.linefollow.user_tag = 0; //not used

    EXOS_ASSERT_OK(exos_dataset_init(&h_ros_topics_typ.linestatus, &h_ros_topics_typ.ros_topics_typ_datamodel, "lineStatus", &h_ros_topics_typ.ext_ros_topics_typ_datamodel.lineStatus.value, sizeof(h_ros_topics_typ.ext_ros_topics_typ_datamodel.lineStatus.value)));
    h_ros_topics_typ.linestatus.user_context = NULL; //not used
    h_ros_topics_typ.linestatus.user_tag = 0; //not used

    return &(h_ros_topics_typ.ext_ros_topics_typ_datamodel);
}
```

- libros_topics_typ.i - SWIG interface file (not shown)

- build.sh - build file shell script (not shown)

- ros_topics_typ.py - Main python script (not shown)

- libros_topics_typ.py - ros_topics_typ python module (not shown)

- _libros_topics_typ.so - ros_topics_typ SWIG library (binary file, 660279 bytes)
### Program Logical/ros_topics_typ/motorCtrl (IEC)

#### motorCtrl.typ - Local data types
```iecst
TYPE
	ros_typ : 	STRUCT
		vel_theta : LREAL;
		vel_x : LREAL;
		r : LREAL;
		cur_theta : LREAL;
		dist : LREAL;
		cur_y : LREAL;
		cur_x : LREAL;
		d_theta : LREAL;
		topics : ros_topics_typ;
		diffLowpassDist : REAL;
		diffDist : LREAL;
		currentLimiter : REAL;
	END_STRUCT;
	local_typ : 	STRUCT
		hw : hw_typ;
		hmi : hmi_typ;
		speed : LREAL;
		encoderOld : INT;
		accLimiter : MTBasicsLimiter;
		PIDCurrent : MTBasicsPID;
		PID : MTBasicsPID;
		distance : LREAL;
		diffEncoder : LREAL;
		filterCurrent : MTFilterMovingAverage;
		filterSpeed : MTFilterMovingAverage;
		diffTime : LREAL;
		timeOld : DINT;
		PIDtune : MTBasicsOscillationTuning;
		lowPass : MTFilterLowPass;
		ton_overcurrent : TON;
		currentLimiter : REAL;
	END_STRUCT;
	hw_typ : 	STRUCT
		input : hw_input_typ;
		output : hw_output_typ;
	END_STRUCT;
	hw_output_typ : 	STRUCT
		pwm : INT;
		clear : BOOL;
	END_STRUCT;
	hw_input_typ : 	STRUCT
		encoder : INT;
		overload : BOOL;
		current : ARRAY[0..7]OF INT;
		nettime : DINT;
	END_STRUCT;
	hmi_typ : 	STRUCT
		config : config_typ;
		output : hmi_output_typ;
		input : hmi_input_typ;
	END_STRUCT;
	hmi_output_typ : 	STRUCT
		current : ARRAY[0..7]OF REAL;
		overload : BOOL;
		distance : LREAL;
		ticks : LREAL;
		currentTotal : REAL;
	END_STRUCT;
	hmi_input_typ : 	STRUCT
		clear : BOOL;
		tune : BOOL;
		resetDistance : BOOL;
	END_STRUCT;
	config_typ : 	STRUCT
		ppm : UDINT := 105860;
		maxCurrent : REAL := 8;
	END_STRUCT;
	common_typ : 	STRUCT
	END_STRUCT;
	suction_typ : 	STRUCT
		valveEnable : BOOL;
		motorEnable : BOOL;
	END_STRUCT;
END_TYPE
```

#### ros_topics_typ.var - ros_topics_typ variable declaration
```iecst
VAR
	config : REFERENCE TO config_typ;
	counter : USINT;
	counter2 : USINT;
	errOld : REAL;
	ExComponentInfo_0 : ExComponentInfo;
	ExDataConnectionInfo_0 : ExDataConnectionInfo;
	ExDatamodelInfo_0 : ExDatamodelInfo;
	ExSyncInfo_0 : ExSyncInfo;
	forwardTimer : TON;
	goalOrientation : REAL;
	hmi : REFERENCE TO hmi_typ;
	hw : REFERENCE TO hw_typ;
	i : USINT;
	iAlive : USINT;
	k : USINT;
	prevBool : BOOL;
	oldOrientation : REAL;
	kd : REAL;
	kp : REAL;
	lastOrientation : REAL;
	lineTest : BOOL;
	localVariables : ARRAY[0..1] OF local_typ;
	mathCheck1 : REAL;
	mathCheck2 : REAL;
	moveForwardTimer : TON;
	remainingOrientation : REAL;
	ros : ros_typ;
	ros_topics_typCyclic_0 : ros_topics_typCyclic;
	ros_topics_typExit_0 : ros_topics_typExit;
	ros_topics_typInit_0 : ros_topics_typInit;
	startOrientation : REAL;
	suction : suction_typ;
	this : REFERENCE TO local_typ;
	turnSwitch : USINT;
	watchIdx : USINT;
END_VAR
```

#### ros_topics_typ.st - ros_topics_typ application
```iecst
PROGRAM _INIT

	ros_topics_typInit_0();

	(* Insert code here *)
	FOR i:=0 TO
		i < 2 BY 1 DO
		setupPointers;

		this.PID.Enable := TRUE;
		this.PID.MinOut := -100;
		this.PID.MaxOut := 100;
		this.PID.PIDParameters.DerivativeTime := 0.00228000456;
		this.PID.PIDParameters.Gain := 78;
		this.PID.PIDParameters.IntegrationTime := 0.02500019;
		this.PID.PIDParameters.FilterTime := 0.000228000456;

		this.PID.Update := TRUE;

		this.PIDCurrent.Enable := TRUE;
		this.PIDCurrent.MinOut := 0;
		this.PIDCurrent.MaxOut := 100;
		this.PIDCurrent.PIDParameters.DerivativeTime := 10;
		this.PIDCurrent.PIDParameters.Gain := 1;
		this.PIDCurrent.PIDParameters.IntegrationTime := 10;
		this.PIDCurrent.PIDParameters.FilterTime := 20;
		this.PIDCurrent.Update := TRUE;
		this.PIDCurrent.SetValue := 8;

		this.filterSpeed.Enable := TRUE;
		this.filterSpeed.WindowLength := 100;
		this.filterSpeed.Update := TRUE;

		this.filterCurrent.Enable := TRUE;
		this.filterCurrent.WindowLength := 3;
		this.filterCurrent.Update := TRUE;

		this.accLimiter.Enable := TRUE;
		this.accLimiter.MaxNegSlewRate := 1;
		this.accLimiter.MaxPosSlewRate := 1;
		this.accLimiter.MaxOut := 1;
		this.accLimiter.MinOut := -1;
		this.accLimiter.Update := TRUE;

		this.PIDtune.SetValue:= 1.0;
		this.PIDtune.MinOut:= 0.0;
		this.PIDtune.MaxOut:= 100.0;
		this.PIDtune.Update := TRUE;

		this.lowPass.Enable := TRUE;
		this.lowPass.CutOffFrequency := 10;
		this.lowPass.Order := 1;
		this.lowPass.Update := TRUE;

		this.encoderOld := this.hw.input.encoder;
		this.timeOld := this.hw.input.nettime;

		this.ton_overcurrent.PT := T#1s;

	END_FOR

END_PROGRAM

PROGRAM _CYCLIC
    //--------------- ex OS ----------------
    //Auto connect:
	ros_topics_typCyclic_0.Enable := ExComponentInfo_0.Operational AND NOT ros_topics_typCyclic_0.Aborted; // Component has been deployed and started up successfully

	//Auto connect when deployment is off and manually started in GPOS:
	//ros_topics_typCyclic_0.Enable := TRUE;
	ros_topics_typCyclic_0.Start := ros_topics_typCyclic_0.Connected;
//	IF counter2 > 5 THEN
//		counter2 := 0;
	ros_topics_typCyclic_0(Handle := ros_topics_typInit_0.Handle, pros_topics_typ := ADR(ros.topics));
//	ELSE
//		counter2 := counter2 + 1;
//	END_IF
	ExComponentInfo_0(ExTargetLink := ADR(gTarget_0), ExComponentLink := ADR(gros_topics_typ_0), Enable := TRUE);

	ExDatamodelInfo_0(ExTargetLink := ADR(gTarget_0), Enable := TRUE, InstanceName := 'ros_topics_typ_0');
	//--------------- ex OS done ----------------
	ExSyncInfo_0(ExTargetLink := ADR(gTarget_0), Enable := TRUE);

	ExDataConnectionInfo_0(ExTargetLink := ADR(gTarget_0),Enable := TRUE);

	forwardTimer();
	moveForwardTimer();
	kp := 0.7;
	kd := 2500;
	suction.motorEnable := ros.topics.vaccumTopic.vaccumMotor;
	suction.valveEnable := ros.topics.vaccumTopic.vaccumValve;
	lineFollow.lineForward := ros.topics.lineFollow.lineForward;
	lineFollow.lineHoldRight := ros.topics.lineFollow.lineHoldRight;
	lineFollow.lineMode := ros.topics.lineFollow.lineMode;
	lineFollow.lineSharpTurn := ros.topics.lineFollow.lineSharpTurn;
	lineFollow.lineInterSection := ros.topics.lineFollow.lineInterSection;
	lineFollow.lineDecision := ros.topics.lineFollow.lineDecision;
	ros.topics.twist.linear.x := MAX(MIN(ros.topics.twist.linear.x,ros.topics.config.maxSpeed),ros.topics.config.minSpeed);
	lineFollow.lineFast := ros.topics.lineFollow.lineFast;
	lineFollow.lineSlow := ros.topics.lineFollow.lineSlow;

	mathCheck1 :=  LREAL_TO_REAL(0.5*(drejMere - errOld)*ros.topics.config.baseWidth/2.0);//LREAL_TO_REAL(0.3-(drejMere*0.35 + 0.01*(drejMere - errOld))*ros.topics.config.baseWidth/2.0);
	mathCheck2 := LREAL_TO_REAL(0.3+(drejMere*0.35 + 0.01*(drejMere-errOld))*ros.topics.config.baseWidth/2.0);

	IF localVariables[0].hmi.output.overload OR localVariables[1].hmi.output.overload OR NOT ros_topics_typCyclic_0.Operational THEN
		IF lineMode THEN

			CASE Test2 OF
				0:
					IF tempDec <> FALSE THEN
						awaitDecision := FALSE;
						tempDec := FALSE;
						orientationReached := TRUE;
					ELSE
						tempDec := lineFollow.lineDecision;
//						sharpTurn  := lineFollow.lineSharpTurn;
//						sammenEnable := lineFollow.lineInterSection;

					END_IF

					localVariables[0].PID.SetValue := 0;
					localVariables[1].PID.SetValue := 0;
				1:

						IF lineFollow.lineSlow THEN
							localVariables[0].PID.SetValue := LREAL_TO_REAL(0.1-((drejMere-errOld)*kp + kd*(errOld)*ros.topics.config.baseWidth/2.0));
							localVariables[1].PID.SetValue := LREAL_TO_REAL(0.1+((drejMere-errOld)*kp + kd*(errOld)*ros.topics.config.baseWidth/2.0));
						ELSIF lineFollow.lineFast THEN
							localVariables[0].PID.SetValue := LREAL_TO_REAL(0.5-((drejMere-errOld)*kp + kd*(errOld)*ros.topics.config.baseWidth/2.0));
							localVariables[1].PID.SetValue := LREAL_TO_REAL(0.5+((drejMere-errOld)*kp + kd*(errOld)*ros.topics.config.baseWidth/2.0));
						ELSE
							localVariables[0].PID.SetValue := LREAL_TO_REAL(0.3-((drejMere-errOld)*kp + kd*(errOld)*ros.topics.config.baseWidth/2.0));
							localVariables[1].PID.SetValue := LREAL_TO_REAL(0.3+((drejMere-errOld)*kp + kd*(errOld)*ros.topics.config.baseWidth/2.0));
						END_IF
					errOld := LREAL_TO_REAL(ros.cur_theta - oldOrientation);
					oldOrientation := LREAL_TO_REAL(ros.cur_theta);
					drejMere := drejMere + errOld;

				2:
					iAlive := iAlive +1;
					orientationReached := FALSE;
					sammenEnable := FALSE;
					lineStatus.lineStatusCode := 70;
					moveForwardTimer.PT := T#3000ms;
					moveForwardTimer.IN := TRUE;
					localVariables[0].PID.SetValue := LREAL_TO_REAL(-((drejMere)*kp*ros.topics.config.baseWidth/2.0));
					localVariables[1].PID.SetValue := LREAL_TO_REAL(((drejMere)*kp*ros.topics.config.baseWidth/2.0));
					IF moveForwardTimer.Q THEN

						moveForwardTimer.IN := FALSE;
						orientationReached := TRUE;
						Test2 := 1;

					END_IF
				-1:
					CASE turnSwitch OF
						0:
							orientationReached := FALSE;
							startOrientation := LREAL_TO_REAL(ros.cur_theta);

							goalOrientation := startOrientation - 0.8929;
							turnSwitch := 5;

						5:
							lastOrientation := LREAL_TO_REAL(ros.cur_theta);
							localVariables[0].PID.SetValue := 0;
							localVariables[1].PID.SetValue := 0;
							IF ros.vel_x = 0 THEN
								forwardTimer.PT := T#1000ms;
								forwardTimer.IN := TRUE;
								IF forwardTimer.Q THEN
									forwardTimer.IN := FALSE;
									turnSwitch := 7;
								END_IF
							END_IF

						7:
							forwardTimer.PT := T#3000ms;
							localVariables[0].PID.SetValue := 0.05;
							localVariables[1].PID.SetValue := 0.05;
							forwardTimer.IN := TRUE;
							IF forwardTimer.Q THEN
								localVariables[0].PID.SetValue := 0;
								localVariables[1].PID.SetValue := 0;
								turnSwitch := 10;
								forwardTimer.IN := FALSE;
							END_IF
						10:

							IF ros.cur_theta + 2.0 < lastOrientation OR ros.cur_theta - 2.0 > lastOrientation THEN
								iAlive := iAlive +1;
								goalOrientation := LREAL_TO_REAL(ros.cur_theta + remainingOrientation);
							ELSIF ros.cur_theta < goalOrientation THEN
								turnSwitch := 20;
							END_IF
							lastOrientation := LREAL_TO_REAL(ros.cur_theta);
							remainingOrientation := LREAL_TO_REAL(goalOrientation - ros.cur_theta);
							localVariables[0].PID.SetValue := -0.05;
							localVariables[1].PID.SetValue := 0.05;

						20:
							localVariables[0].PID.SetValue := 0;
							localVariables[1].PID.SetValue := 0;

							turnSwitch := 21;

						21:
							ros.topics.lineStatus.lineStatusCode := 50;
							IF moveForward <> TRUE THEN
								orientationReached := TRUE;
								turnSwitch := 0;
								Test2 := 10;
							END_IF
					END_CASE
				5:
					errOld := 0;
					oldOrientation := 0;
					IF moveForward THEN
						lineStatus.lineStatusCode := 90;
						localVariables[0].PID.SetValue := 0.1;
						localVariables[1].PID.SetValue := 0.1;
						moveForwardTimer.PT := T#5000ms;
						moveForwardTimer.IN := TRUE;
						IF moveForwardTimer.Q THEN
							localVariables[0].PID.SetValue := 0.1;
							localVariables[1].PID.SetValue := 0.1;
							//Test2 := 10;
							moveForwardTimer.IN := FALSE;
						END_IF
					ELSE
						Test2 := 10;
					END_IF

				10:
					lineStatus.lineStatusCode := 90;
					localVariables[0].PID.SetValue := LREAL_TO_REAL(-(drejMere*0.45)*ros.topics.config.baseWidth/2.0);
					localVariables[1].PID.SetValue := LREAL_TO_REAL((drejMere*0.45)*ros.topics.config.baseWidth/2.0);
					moveForwardTimer.IN := FALSE;
				20:
					CASE turnSwitch OF
						0:
							orientationReached := FALSE;
							startOrientation := LREAL_TO_REAL(ros.cur_theta);
							IF rightTurn THEN
								goalOrientation := startOrientation - 1.4929;
								turnSwitch := 5;
							ELSE
								goalOrientation := startOrientation + 1.4929;
								turnSwitch := 5;
							END_IF

						5:
							lastOrientation := LREAL_TO_REAL(ros.cur_theta);
							localVariables[0].PID.SetValue := 0;
							localVariables[1].PID.SetValue := 0;
							IF ros.vel_x = 0 THEN
								turnSwitch := 7;
							END_IF

						7:
							forwardTimer.PT := T#5000ms;
							localVariables[0].PID.SetValue := 0.05;
							localVariables[1].PID.SetValue := 0.05;
							forwardTimer.IN := TRUE;
							IF forwardTimer.Q THEN
								localVariables[0].PID.SetValue := 0;
								localVariables[1].PID.SetValue := 0;
								turnSwitch := 10;
								forwardTimer.IN := FALSE;
							END_IF
						10:

							IF ros.cur_theta + 2.0 < lastOrientation OR ros.cur_theta - 2.0 > lastOrientation THEN
								iAlive := iAlive +1;
								goalOrientation := LREAL_TO_REAL(ros.cur_theta + remainingOrientation);
							ELSIF rightTurn THEN
								IF ros.cur_theta < goalOrientation THEN
									turnSwitch := 20;
								END_IF
							ELSIF ros.cur_theta > goalOrientation THEN
								turnSwitch := 20;
							END_IF
							lastOrientation := LREAL_TO_REAL(ros.cur_theta);
							remainingOrientation := LREAL_TO_REAL(goalOrientation - ros.cur_theta);
							IF rightTurn THEN
								localVariables[0].PID.SetValue := -0.05;
								localVariables[1].PID.SetValue := 0.05;
							ELSE
								localVariables[0].PID.SetValue := 0.05;
								localVariables[1].PID.SetValue := -0.05;
								END_IF
						20:
							orientationReached := TRUE;
							localVariables[0].PID.SetValue := 0;
							localVariables[1].PID.SetValue := 0;
							sharpTurn := FALSE;
							Test2 := 10;
							turnSwitch := 0;
					END_CASE

			END_CASE
		ELSE
		localVariables[0].PID.SetValue := 0;
		localVariables[1].PID.SetValue := 0;
		END_IF
	/////////////////////////////// EXOS DEAKTIVERET ///////////////////////////////////////////////////////////////
	/////////////////////////////// EXOS AKTIVERET//////////////////////////////////////////////////////////////////

	ELSE
		IF ros.topics.lineFollow.lineMode THEN

			CASE Test2 OF
				0:
					iAlive := iAlive +1;
					IF tempDec <> FALSE THEN
						awaitDecision := FALSE;
						tempDec := FALSE;
						orientationReached := TRUE;
						lineStatus.lineStatusCode := 20;

					ELSE

						tempDec := lineFollow.lineDecision;
						sharpTurn  := lineFollow.lineSharpTurn;
						sammenEnable := lineFollow.lineInterSection;
						lineStatus.lineStatusCode := 20;

					END_IF

					localVariables[0].PID.SetValue := 0;
					localVariables[1].PID.SetValue := 0;
				1:
					//iAlive := iAlive +1;
					IF lineFollow.lineSlow THEN
						localVariables[0].PID.SetValue := LREAL_TO_REAL(0.1-((drejMere-errOld)*kp + kd*(errOld)*ros.topics.config.baseWidth/2.0));
						localVariables[1].PID.SetValue := LREAL_TO_REAL(0.1+((drejMere-errOld)*kp + kd*(errOld)*ros.topics.config.baseWidth/2.0));
					ELSIF lineFollow.lineFast THEN
						localVariables[0].PID.SetValue := LREAL_TO_REAL(0.5-((drejMere-errOld)*kp + kd*(errOld)*ros.topics.config.baseWidth/2.0));
						localVariables[1].PID.SetValue := LREAL_TO_REAL(0.5+((drejMere-errOld)*kp + kd*(errOld)*ros.topics.config.baseWidth/2.0));
					ELSE
						localVariables[0].PID.SetValue := LREAL_TO_REAL(0.3-((drejMere-errOld)*kp + kd*(errOld)*ros.topics.config.baseWidth/2.0));
						localVariables[1].PID.SetValue := LREAL_TO_REAL(0.3+((drejMere-errOld)*kp + kd*(errOld)*ros.topics.config.baseWidth/2.0));
					END_IF
					errOld := LREAL_TO_REAL(ros.cur_theta - oldOrientation);
					oldOrientation := LREAL_TO_REAL(ros.cur_theta);
					drejMere := drejMere + errOld;

				2:
					orientationReached := FALSE;
					lineStatus.lineStatusCode := 70;
					moveForwardTimer.PT := T#3000ms;
					moveForwardTimer.IN := TRUE;
					localVariables[0].PID.SetValue := LREAL_TO_REAL(0.1-((drejMere)*kp*ros.topics.config.baseWidth/2.0));
					localVariables[1].PID.SetValue := LREAL_TO_REAL(0.1+((drejMere)*kp*ros.topics.config.baseWidth/2.0));

					IF moveForwardTimer.Q THEN
						orientationReached := TRUE;
						moveForwardTimer.IN := FALSE;

					END_IF
				-1:

					CASE turnSwitch OF
						0:
							orientationReached := FALSE;
							startOrientation := LREAL_TO_REAL(ros.cur_theta);

							goalOrientation := startOrientation - 1.4929;
							turnSwitch := 5;

						5:
							lastOrientation := LREAL_TO_REAL(ros.cur_theta);
							localVariables[0].PID.SetValue := 0;
							localVariables[1].PID.SetValue := 0;
							IF ros.vel_x = 0 THEN
								forwardTimer.PT := T#1000ms;
								forwardTimer.IN := TRUE;
								IF forwardTimer.Q THEN
									forwardTimer.IN := FALSE;
									turnSwitch := 7;
								END_IF
							END_IF

						7:
							forwardTimer.PT := T#3000ms;
							localVariables[0].PID.SetValue := 0.05;
							localVariables[1].PID.SetValue := 0.05;
							forwardTimer.IN := TRUE;
							IF forwardTimer.Q THEN
								localVariables[0].PID.SetValue := 0;
								localVariables[1].PID.SetValue := 0;
								turnSwitch := 10;
								forwardTimer.IN := FALSE;
							END_IF
						10:

							IF ros.cur_theta + 2.0 < lastOrientation OR ros.cur_theta - 2.0 > lastOrientation THEN
								goalOrientation := LREAL_TO_REAL(ros.cur_theta + remainingOrientation);
							ELSIF ros.cur_theta < goalOrientation THEN
								turnSwitch := 20;
							END_IF
							lastOrientation := LREAL_TO_REAL(ros.cur_theta);
							remainingOrientation := LREAL_TO_REAL(goalOrientation - ros.cur_theta);
							localVariables[0].PID.SetValue := -0.05;
							localVariables[1].PID.SetValue := 0.05;

						20:

							lineStatus.lineStatusCode := 50;
							localVariables[0].PID.SetValue := 0;
							localVariables[1].PID.SetValue := 0;

							turnSwitch := 21;
						21:
							lineStatus.lineStatusCode := 50;
							localVariables[0].PID.SetValue := 0;
							localVariables[1].PID.SetValue := 0;
							IF TRUE <> ros.topics.lineFollow.lineForward THEN
								orientationReached := TRUE;
								turnSwitch := 0;
								Test2 := 10;
							END_IF
					END_CASE

				5:
					errOld := 0;
					oldOrientation := 0;
					IF lineFollow.lineForward THEN
						lineStatus.lineStatusCode := 90;
						localVariables[0].PID.SetValue := 0.1;
						localVariables[1].PID.SetValue := 0.1;
						moveForwardTimer.PT := T#5000ms;
						moveForwardTimer.IN := TRUE;
						IF moveForwardTimer.Q THEN
							localVariables[0].PID.SetValue := 0;
							localVariables[1].PID.SetValue := 0;
							Test2 := 10;
							moveForwardTimer.IN := FALSE;
						END_IF

					ELSE
						Test2 := 10;
					END_IF

				10:
					lineStatus.lineStatusCode := 90;
					localVariables[0].PID.SetValue := LREAL_TO_REAL(-(drejMere*0.45)*ros.topics.config.baseWidth/2.0);
					localVariables[1].PID.SetValue := LREAL_TO_REAL((drejMere*0.45)*ros.topics.config.baseWidth/2.0);
					moveForwardTimer.IN := FALSE;
				20:
					CASE turnSwitch OF
						0:
							lineStatus.lineStatusCode := 20;
							orientationReached := FALSE;
							startOrientation := LREAL_TO_REAL(ros.cur_theta);
							IF rightTurn THEN
								goalOrientation := startOrientation - 1.4929;
								turnSwitch := 5;
							ELSE
								goalOrientation := startOrientation + 1.4929;
								turnSwitch := 5;
							END_IF

						5:
							lastOrientation := LREAL_TO_REAL(ros.cur_theta);
							localVariables[0].PID.SetValue := 0;
							localVariables[1].PID.SetValue := 0;
							IF ros.vel_x = 0 THEN
								turnSwitch := 7;
							END_IF

						7:
							forwardTimer.PT := T#5000ms;
							localVariables[0].PID.SetValue := 0.05;
							localVariables[1].PID.SetValue := 0.05;
							forwardTimer.IN := TRUE;
							IF forwardTimer.Q THEN
								localVariables[0].PID.SetValue := 0;
								localVariables[1].PID.SetValue := 0;
								turnSwitch := 10;
								forwardTimer.IN := FALSE;
							END_IF
						10:

							IF ros.cur_theta + 2.0 < lastOrientation OR ros.cur_theta - 2.0 > lastOrientation THEN
								goalOrientation := LREAL_TO_REAL(ros.cur_theta + remainingOrientation);
							ELSIF rightTurn THEN
								IF ros.cur_theta < goalOrientation THEN
									turnSwitch := 20;
								END_IF
							ELSIF ros.cur_theta > goalOrientation THEN
								turnSwitch := 20;
							END_IF
							lastOrientation := LREAL_TO_REAL(ros.cur_theta);
							remainingOrientation := LREAL_TO_REAL(goalOrientation - ros.cur_theta);
							IF rightTurn THEN
								localVariables[0].PID.SetValue := -0.05;
								localVariables[1].PID.SetValue := 0.05;
							ELSE
								localVariables[0].PID.SetValue := 0.05;
								localVariables[1].PID.SetValue := -0.05;
							END_IF
						20:
							orientationReached := TRUE;
							localVariables[0].PID.SetValue := 0;
							localVariables[1].PID.SetValue := 0;
							sharpTurn := FALSE;
							Test2 := 10;
							turnSwitch := 0;
					END_CASE

			END_CASE
		ELSE

			localVariables[0].PID.SetValue := LREAL_TO_REAL(ros.topics.twist.linear.x + ros.topics.twist.angular.z * ros.topics.config.baseWidth / 2.0) * ros.currentLimiter;  // m/s
			localVariables[1].PID.SetValue := LREAL_TO_REAL(ros.topics.twist.linear.x - ros.topics.twist.angular.z * ros.topics.config.baseWidth / 2.0) * ros.currentLimiter;
		END_IF
	END_IF

	FOR i:=0 TO 1 BY 1 DO
		setupPointers;

		hmi.output.overload := FALSE;

		hmi.output.currentTotal := 0;

		FOR k:=0 TO 7 DO

			hmi.output.current[k] := INT_TO_REAL(hw.input.current[k])*10.0/32767.0;
			hmi.output.currentTotal := hmi.output.currentTotal + hmi.output.current[k];
		END_FOR

		hmi.output.currentTotal := hmi.output.currentTotal /2.0;

		IF this.filterCurrent.UpdateDone THEN
			this.filterSpeed.Update := FALSE;
		END_IF

		this.filterCurrent(In := hmi.output.currentTotal);

		IF this.PIDCurrent.UpdateDone THEN
			this.PIDCurrent.Update := FALSE;
		END_IF

		this.PIDCurrent(ActValue := this.filterCurrent.Out);

		this.currentLimiter := 1;//this.PIDCurrent.Out/100;

		hmi.output.overload := hw.input.overload;

		this.ton_overcurrent(IN := hmi.output.overload);
		IF this.ton_overcurrent.Q THEN
			this.hmi.input.clear := TRUE;
		END_IF

		hw.output.clear := hmi.input.clear;

		IF NOT hmi.output.overload THEN
			hmi.input.clear := FALSE;
		END_IF

		this.diffTime := DINT_TO_LREAL(hw.input.nettime -this.timeOld);
		IF this.diffTime < -100000.0 THEN
			this.diffTime := this.diffTime + 2*2147483647;
		END_IF
		this.diffTime := this.diffTime /1000.0;
		this.timeOld := hw.input.nettime;

		this.diffEncoder := INT_TO_LREAL(hw.input.encoder)-INT_TO_LREAL(this.encoderOld);

		this.encoderOld := hw.input.encoder;

		IF this.diffEncoder > 32727 THEN

			this.diffEncoder := this.diffEncoder - 2*32767;

		ELSIF this.diffEncoder < -32727 THEN

			this.diffEncoder := this.diffEncoder + 2*32767;

		END_IF

		hmi.output.ticks := hmi.output.ticks + this.diffEncoder;
		hmi.output.distance := hmi.output.ticks / UDINT_TO_LREAL(config.ppm);

		IF hmi.input.resetDistance THEN
			hmi.input.resetDistance := FALSE;
			hmi.output.ticks := 0;
			hmi.output.distance := 0;
		END_IF

		this.distance 	:= this.diffEncoder/UDINT_TO_LREAL(config.ppm);

		this.lowPass.In := LREAL_TO_REAL(this.distance);
		this.lowPass();

		this.speed 		:= this.distance * 1000/this.diffTime;

		IF this.filterSpeed.UpdateDone THEN
			this.filterSpeed.Update := FALSE;
		END_IF

		this.filterSpeed(In := LREAL_TO_REAL(this.speed));

		IF this.accLimiter.UpdateDone THEN
			this.accLimiter.Update := FALSE;
		END_IF

		this.accLimiter(In := this.PID.SetValue);

		IF this.PID.UpdateDone THEN
			this.PID.Update := FALSE;
		END_IF

		this.PID.ActValue := LREAL_TO_REAL(this.speed);
		this.PID.SetValue := this.accLimiter.Out;
		// PID TUNE

		IF hmi.input.tune THEN
			this.PIDtune.Enable := TRUE;
		END_IF

		this.PIDtune.ActValue := LREAL_TO_REAL(this.speed);

		IF this.PIDtune.TuningDone THEN
			this.PIDtune.Start := FALSE;
			this.PID.IntegrationPartPresetValue := this.PIDtune.Out;
			this.PID.SetIntegrationPart := TRUE;
		ELSIF this.PIDtune.Active AND NOT this.PIDtune.Update THEN
			//	this.PIDtune.Start := TRUE;
		END_IF

		IF this.PIDtune.UpdateDone THEN
			this.PIDtune.Update := FALSE;
		END_IF

		(* call function block *)
		this.PID();
		this.PIDtune();

		this.PID.SetIntegrationPart := FALSE;

		IF hmi.input.tune THEN
			hw.output.pwm := REAL_TO_INT(this.PIDtune.Out*327.67);
		ELSE
			hw.output.pwm := REAL_TO_INT(this.PID.Out*327.67);
		END_IF

	END_FOR

	ros.currentLimiter := MIN(localVariables[0].currentLimiter,localVariables[1].currentLimiter);

	ros.diffDist := localVariables[1].distance-localVariables[0].distance;
	ros.diffLowpassDist := localVariables[1].lowPass.Out-localVariables[0].lowPass.Out;

	ros.dist := (localVariables[1].distance+localVariables[0].distance)/2;

	IF localVariables[0].diffEncoder = localVariables[1].diffEncoder THEN
		ros.d_theta := 0.0;
		ros.cur_x := ros.cur_x + ros.dist * COS(ros.cur_theta);
		ros.cur_y := ros.cur_y + ros.dist * SIN(ros.cur_theta);
	ELSE
		ros.d_theta := -(localVariables[1].distance - localVariables[0].distance) / ros.topics.config.baseWidth;
		ros.dist := (localVariables[1].distance+localVariables[0].distance)/2;
		ros.r := ros.dist / ros.d_theta;
		ros.cur_x := ros.cur_x + ros.r * (SIN(ros.d_theta + ros.cur_theta) - SIN(ros.cur_theta));
		ros.cur_y := ros.cur_y - ros.r * (COS(ros.d_theta + ros.cur_theta) - COS(ros.cur_theta));
		ros.cur_theta := normalizeAngle(ros.cur_theta + ros.d_theta);
	END_IF

	ros.vel_x := ros.dist * (1000.0/localVariables[0].diffTime);
	ros.vel_theta := ros.d_theta * (1000.0/localVariables[0].diffTime);

	// set ros data

	IF lineStatus.lineStatusCode = 0 THEN
		evaluateStatus;
	END_IF

//	IF counter > 5  THEN
//		counter := 0;
	ros.topics.odemetry.pose.pose.position.x 	:= ros.cur_x;
	ros.topics.odemetry.pose.pose.position.y	:= ros.cur_y;
	ros.topics.odemetry.pose.pose.orientation.z	:= ros.cur_theta;

	ros.topics.odemetry.twist.twist.linear.x  	:= ros.vel_x;
	ros.topics.odemetry.twist.twist.angular.z 	:= ros.vel_theta;
	IF ros.topics.lineStatus.lineStatusCode <> lineStatus.lineStatusCode THEN //AND lineFollow.lineMode THEN
		ros.topics.lineStatus.lineStatusCode := lineStatus.lineStatusCode;
	END_IF
//	ELSE
//		counter := counter +1;
//	END_IF
	lineStatus.lineStatusCode := 0;
	setupWatchPointers;

END_PROGRAM

PROGRAM _EXIT

	ros_topics_typExit_0(Handle := ros_topics_typInit_0.Handle);

END_PROGRAM
```

### Library Logical/ros_topics_typ/ros_topics (ANSIC)
Depends on: ExData

#### ros_topics_typ.typ - ros_topics_typ datamodel declaration
```iecst
TYPE
	ros_topic_point_typ : 	STRUCT  (*this expresses velocity in free space broken into its linear and angular parts.*)
		y : LREAL;
		z : LREAL;
		x : LREAL;
	END_STRUCT;
	ros_topic_vector3_typ : 	STRUCT  (*this expresses velocity in free space broken into its linear and angular parts.*)
		y : LREAL;
		z : LREAL;
		x : LREAL;
	END_STRUCT;
	ros_topic_twist_typ : 	STRUCT  (*This expresses velocity in free space broken into its linear and angular parts.*)
		angular : ros_topic_vector3_typ;
		linear : ros_topic_vector3_typ;
	END_STRUCT;
	ros_topic_twistCor_typ : 	STRUCT  (*This expresses velocity in free space with uncertainty.*)
		twist : ros_topic_twist_typ;
	END_STRUCT;
	ros_topic_quaternion_typ : 	STRUCT  (*This represents an orientation in free space in quaternion form.*)
		y : LREAL;
		z : LREAL;
		w : LREAL;
		x : LREAL;
	END_STRUCT;
	ros_topic_odemety_point_typ : 	STRUCT  (*This contains the position of a point in free space*)
		y : LREAL;
		z : LREAL;
		x : LREAL;
	END_STRUCT;
	ros_topic_pose_typ : 	STRUCT  (*A representation of pose in free space, composed of position and orientation. *)
		position : ros_topic_point_typ;
		orientation : ros_topic_quaternion_typ;
	END_STRUCT;
	ros_topic_poseCor_typ : 	STRUCT  (*This represents a pose in free space with uncertainty.*)
		pose : ros_topic_pose_typ;
	END_STRUCT;
	ros_topic_time_typ : 	STRUCT
		nsec : UDINT;
		sec : UDINT;
	END_STRUCT;
	ros_topic_header_typ : 	STRUCT
		stamp : ros_topic_time_typ;
		seq : UDINT;
		frame_id : STRING[20];
	END_STRUCT;
	ros_topic_odemety_typ : 	STRUCT
		pose : ros_topic_poseCor_typ;
		twist : ros_topic_twistCor_typ;
		header : ros_topic_header_typ;
	END_STRUCT;
	ros_config_typ : 	STRUCT
		maxSpeed : LREAL := 2;
		minSpeed : LREAL := -2;
		baseWidth : LREAL := 0.308;
	END_STRUCT;
	ros_topics_typ : 	STRUCT
		odemetry : ros_topic_odemety_typ; (*PUB*)
		twist : ros_topic_twist_typ; (*SUB*)
		config : ros_config_typ; (*SUB*)
		encoder : ros_encoder; (*PUB*)
		vaccumTopic : ros_armBools; (*SUB*)
		lineFollow : ros_lineMode; (*SUB*)
		lineStatus : ros_lineStatus; (*PUB*)
	END_STRUCT;
	ros_motorCtrl : 	STRUCT
		twist : ros_topic_twist_typ; (*SUB*)
		config : ros_config_typ; (*SUB*)
	END_STRUCT;
	ros_encoder : 	STRUCT
		encoder1 : INT;
		encoder2 : INT;
	END_STRUCT;
	ros_armBools : 	STRUCT
		vaccumValve : BOOL;
		vaccumMotor : BOOL;
	END_STRUCT;
	ros_lineMode : 	STRUCT
		lineMode : BOOL;
		lineSharpTurn : BOOL;
		lineHoldRight : BOOL;
		lineForward : BOOL;
		lineInterSection : BOOL;
		lineDecision : BOOL;
		lineFast : BOOL;
		lineSlow : BOOL;
	END_STRUCT;
	ros_lineStatus : 	STRUCT
		lineStatusCode : INT;
	END_STRUCT;
END_TYPE
```

#### exos_ros_topics_typ.c - Generated datamodel source for ros_topics_typ
```c
/*Automatically generated c file from ros_topics_typ.typ*/

#include "exos_ros_topics_typ.h"

const char config_ros_topics_typ[] = "{\"name\":\"struct\",\"attributes\":{\"name\":\"<NAME>\",\"dataType\":\"ros_topics_typ\",\"info\":\"<infoId0>\"},\"children\":[{\"name\":\"struct\",\"attributes\":{\"name\":\"odemetry\",\"dataType\":\"ros_topic_odemety_typ\",\"comment\":\"PUB\",\"info\":\"<infoId1>\"},\"children\":[{\"name\":\"struct\",\"attributes\":{\"name\":\"pose\",\"dataType\":\"ros_topic_poseCor_typ\",\"info\":\"<infoId2>\"},\"children\":[{\"name\":\"struct\",\"attributes\":{\"name\":\"pose\",\"dataType\":\"ros_topic_pose_typ\",\"info\":\"<infoId3>\"},\"children\":[{\"name\":\"struct\",\"attributes\":{\"name\":\"position\",\"dataType\":\"ros_topic_point_typ\",\"info\":\"<infoId4>\"},\"children\":[{\"name\":\"variable\",\"attributes\":{\"name\":\"y\",\"dataType\":\"LREAL\",\"info\":\"<infoId5>\"}},{\"name\":\"variable\",\"attributes\":{\"name\":\"z\",\"dataType\":\"LREAL\",\"info\":\"<infoId6>\"}},{\"name\":\"variable\",\"attributes\":{\"name\":\"x\",\"dataType\":\"LREAL\",\"info\":\"<infoId7>\"}}]},{\"name\":\"struct\",\"attributes\":{\"name\":\"orientation\",\"dataType\":\"ros_topic_quaternion_typ\",\"info\":\"<infoId8>\"},\"children\":[{\"name\":\"variable\",\"attributes\":{\"name\":\"y\",\"dataType\":\"LREAL\",\"info\":\"<infoId9>\"}},{\"name\":\"variable\",\"attributes\":{\"name\":\"z\",\"dataType\":\"LREAL\",\"info\":\"<infoId10>\"}},{\"name\":\"variable\",\"attributes\":{\"name\":\"w\",\"dataType\":\"LREAL\",\"info\":\"<infoId11>\"}},{\"name\":\"variable\",\"attributes\":{\"name\":\"x\",\"dataType\":\"LREAL\",\"info\":\"<infoId12>\"}}]}]}]},{\"name\":\"struct\",\"attributes\":{\"name\":\"twist\",\"dataType\":\"ros_topic_twistCor_typ\",\"info\":\"<infoId13>\"},\"children\":[{\"name\":\"struct\",\"attributes\":{\"name\":\"twist\",\"dataType\":\"ros_topic_twist_typ\",\"info\":\"<infoId14>\"},\"children\":[{\"name\":\"struct\",\"attributes\":{\"name\":\"angular\",\"dataType\":\"ros_topic_vector3_typ\",\"info\":\"<infoId15>\"},\"children\":[{\"name\":\"variable\",\"attributes\":{\"name\":\"y\",\"dataType\":\"LREAL\",\"info\":\"<infoId16>\"}},{\"name\":\"variable\",\"attributes\":{\"name\":\"z\",\"dataType\":\"LREAL\",\"info\":\"<infoId17>\"}},{\"name\":\"variable\",\"attributes\":{\"name\":\"x\",\"dataType\":\"LREAL\",\"info\":\"<infoId18>\"}}]},{\"name\":\"struct\",\"attributes\":{\"name\":\"linear\",\"dataType\":\"ros_topic_vector3_typ\",\"info\":\"<infoId19>\"},\"children\":[{\"name\":\"variable\",\"attributes\":{\"name\":\"y\",\"dataType\":\"LREAL\",\"info\":\"<infoId20>\"}},{\"name\":\"variable\",\"attributes\":{\"name\":\"z\",\"dataType\":\"LREAL\",\"info\":\"<infoId21>\"}},{\"name\":\"variable\",\"attributes\":{\"name\":\"x\",\"dataType\":\"LREAL\",\"info\":\"<infoId22>\"}}]}]}]},{\"name\":\"struct\",\"attributes\":{\"name\":\"header\",\"dataType\":\"ros_topic_header_typ\",\"info\":\"<infoId23>\"},\"children\":[{\"name\":\"struct\",\"attributes\":{\"name\":\"stamp\",\"dataType\":\"ros_topic_time_typ\",\"info\":\"<infoId24>\"},\"children\":[{\"name\":\"variable\",\"attributes\":{\"name\":\"nsec\",\"dataType\":\"UDINT\",\"info\":\"<infoId25>\"}},{\"name\":\"variable\",\"attributes\":{\"name\":\"sec\",\"dataType\":\"UDINT\",\"info\":\"<infoId26>\"}}]},{\"name\":\"variable\",\"attributes\":{\"name\":\"seq\",\"dataType\":\"UDINT\",\"info\":\"<infoId27>\"}},{\"name\":\"variable\",\"attributes\":{\"name\":\"frame_id\",\"dataType\":\"STRING\",\"stringLength\":21,\"info\":\"<infoId28>\"}}]}]},{\"name\":\"struct\",\"attributes\":{\"name\":\"twist\",\"dataType\":\"ros_topic_twist_typ\",\"comment\":\"SUB\",\"info\":\"<infoId29>\"},\"children\":[{\"name\":\"struct\",\"attributes\":{\"name\":\"angular\",\"dataType\":\"ros_topic_vector3_typ\",\"info\":\"<infoId30>\"},\"children\":[{\"name\":\"variable\",\"attributes\":{\"name\":\"y\",\"dataType\":\"LREAL\",\"info\":\"<infoId31>\"}},{\"name\":\"variable\",\"attributes\":{\"name\":\"z\",\"dataType\":\"LREAL\",\"info\":\"<infoId32>\"}},{\"name\":\"variable\",\"attributes\":{\"name\":\"x\",\"dataType\":\"LREAL\",\"info\":\"<infoId33>\"}}]},{\"name\":\"struct\",\"attributes\":{\"name\":\"linear\",\"dataType\":\"ros_topic_vector3_typ\",\"info\":\"<infoId34>\"},\"children\":[{\"name\":\"variable\",\"attributes\":{\"name\":\"y\",\"dataType\":\"LREAL\",\"info\":\"<infoId35>\"}},{\"name\":\"variable\",\"attributes\":{\"name\":\"z\",\"dataType\":\"LREAL\",\"info\":\"<infoId36>\"}},{\"name\":\"variable\",\"attributes\":{\"name\":\"x\",\"dataType\":\"LREAL\",\"info\":\"<infoId37>\"}}]}]},{\"name\":\"struct\",\"attributes\":{\"name\":\"config\",\"dataType\":\"ros_config_typ\",\"comment\":\"SUB\",\"info\":\"<infoId38>\"},\"children\":[{\"name\":\"variable\",\"attributes\":{\"name\":\"maxSpeed\",\"dataType\":\"LREAL\",\"info\":\"<infoId39>\"}},{\"name\":\"variable\",\"attributes\":{\"name\":\"minSpeed\",\"dataType\":\"LREAL\",\"info\":\"<infoId40>\"}},{\"name\":\"variable\",\"attributes\":{\"name\":\"baseWidth\",\"dataType\":\"LREAL\",\"info\":\"<infoId41>\"}}]},{\"name\":\"struct\",\"attributes\":{\"name\":\"encoder\",\"dataType\":\"ros_encoder\",\"comment\":\"PUB\",\"info\":\"<infoId42>\"},\"children\":[{\"name\":\"variable\",\"attributes\":{\"name\":\"encoder1\",\"dataType\":\"INT\",\"info\":\"<infoId43>\"}},{\"name\":\"variable\",\"attributes\":{\"name\":\"encoder2\",\"dataType\":\"INT\",\"info\":\"<infoId44>\"}}]},{\"name\":\"struct\",\"attributes\":{\"name\":\"vaccumTopic\",\"dataType\":\"ros_armBools\",\"comment\":\"SUB\",\"info\":\"<infoId45>\"},\"children\":[{\"name\":\"variable\",\"attributes\":{\"name\":\"vaccumValve\",\"dataType\":\"BOOL\",\"info\":\"<infoId46>\"}},{\"name\":\"variable\",\"attributes\":{\"name\":\"vaccumMotor\",\"dataType\":\"BOOL\",\"info\":\"<infoId47>\"}}]},{\"name\":\"struct\",\"attributes\":{\"name\":\"lineFollow\",\"dataType\":\"ros_lineMode\",\"comment\":\"SUB\",\"info\":\"<infoId48>\"},\"children\":[{\"name\":\"variable\",\"attributes\":{\"name\":\"lineMode\",\"dataType\":\"BOOL\",\"info\":\"<infoId49>\"}},{\"name\":\"variable\",\"attributes\":{\"name\":\"lineSharpTurn\",\"dataType\":\"BOOL\",\"info\":\"<infoId50>\"}},{\"name\":\"variable\",\"attributes\":{\"name\":\"lineHoldRight\",\"dataType\":\"BOOL\",\"info\":\"<infoId51>\"}},{\"name\":\"variable\",\"attributes\":{\"name\":\"lineForward\",\"dataType\":\"BOOL\",\"info\":\"<infoId52>\"}},{\"name\":\"variable\",\"attributes\":{\"name\":\"lineInterSection\",\"dataType\":\"BOOL\",\"info\":\"<infoId53>\"}},{\"name\":\"variable\",\"attributes\":{\"name\":\"lineDecision\",\"dataType\":\"BOOL\",\"info\":\"<infoId54>\"}},{\"name\":\"variable\",\"attributes\":{\"name\":\"lineFast\",\"dataType\":\"BOOL\",\"info\":\"<infoId55>\"}},{\"name\":\"variable\",\"attributes\":{\"name\":\"lineSlow\",\"dataType\":\"BOOL\",\"info\":\"<infoId56>\"}}]},{\"name\":\"struct\",\"attributes\":{\"name\":\"lineStatus\",\"dataType\":\"ros_lineStatus\",\"comment\":\"PUB\",\"info\":\"<infoId57>\"},\"children\":[{\"name\":\"variable\",\"attributes\":{\"name\":\"lineStatusCode\",\"dataType\":\"INT\",\"info\":\"<infoId58>\"}}]}]}";

/*Connect the ros_topics_typ datamodel to the server*/
EXOS_ERROR_CODE exos_datamodel_connect_ros_topics_typ(exos_datamodel_handle_t *datamodel, exos_datamodel_event_cb datamodel_event_callback)
{
    ros_topics_typ data;
    exos_dataset_info_t datasets[] = {
        {EXOS_DATASET_BROWSE_NAME_INIT,{}},
        {EXOS_DATASET_BROWSE_NAME(odemetry),{}},
        {EXOS_DATASET_BROWSE_NAME(odemetry.pose),{}},
        {EXOS_DATASET_BROWSE_NAME(odemetry.pose.pose),{}},
        {EXOS_DATASET_BROWSE_NAME(odemetry.pose.pose.position),{}},
        {EXOS_DATASET_BROWSE_NAME(odemetry.pose.pose.position.y),{}},
        {EXOS_DATASET_BROWSE_NAME(odemetry.pose.pose.position.z),{}},
        {EXOS_DATASET_BROWSE_NAME(odemetry.pose.pose.position.x),{}},
        {EXOS_DATASET_BROWSE_NAME(odemetry.pose.pose.orientation),{}},
        {EXOS_DATASET_BROWSE_NAME(odemetry.pose.pose.orientation.y),{}},
        {EXOS_DATASET_BROWSE_NAME(odemetry.pose.pose.orientation.z),{}},
        {EXOS_DATASET_BROWSE_NAME(odemetry.pose.pose.orientation.w),{}},
        {EXOS_DATASET_BROWSE_NAME(odemetry.pose.pose.orientation.x),{}},
        {EXOS_DATASET_BROWSE_NAME(odemetry.twist),{}},
        {EXOS_DATASET_BROWSE_NAME(odemetry.twist.twist),{}},
        {EXOS_DATASET_BROWSE_NAME(odemetry.twist.twist.angular),{}},
        {EXOS_DATASET_BROWSE_NAME(odemetry.twist.twist.angular.y),{}},
        {EXOS_DATASET_BROWSE_NAME(odemetry.twist.twist.angular.z),{}},
        {EXOS_DATASET_BROWSE_NAME(odemetry.twist.twist.angular.x),{}},
        {EXOS_DATASET_BROWSE_NAME(odemetry.twist.twist.linear),{}},
        {EXOS_DATASET_BROWSE_NAME(odemetry.twist.twist.linear.y),{}},
        {EXOS_DATASET_BROWSE_NAME(odemetry.twist.twist.linear.z),{}},
        {EXOS_DATASET_BROWSE_NAME(odemetry.twist.twist.linear.x),{}},
        {EXOS_DATASET_BROWSE_NAME(odemetry.header),{}},
        {EXOS_DATASET_BROWSE_NAME(odemetry.header.stamp),{}},
        {EXOS_DATASET_BROWSE_NAME(odemetry.header.stamp.nsec),{}},
        {EXOS_DATASET_BROWSE_NAME(odemetry.header.stamp.sec),{}},
        {EXOS_DATASET_BROWSE_NAME(odemetry.header.seq),{}},
        {EXOS_DATASET_BROWSE_NAME(odemetry.header.frame_id),{}},
        {EXOS_DATASET_BROWSE_NAME(twist),{}},
        {EXOS_DATASET_BROWSE_NAME(twist.angular),{}},
        {EXOS_DATASET_BROWSE_NAME(twist.angular.y),{}},
        {EXOS_DATASET_BROWSE_NAME(twist.angular.z),{}},
        {EXOS_DATASET_BROWSE_NAME(twist.angular.x),{}},
        {EXOS_DATASET_BROWSE_NAME(twist.linear),{}},
        {EXOS_DATASET_BROWSE_NAME(twist.linear.y),{}},
        {EXOS_DATASET_BROWSE_NAME(twist.linear.z),{}},
        {EXOS_DATASET_BROWSE_NAME(twist.linear.x),{}},
        {EXOS_DATASET_BROWSE_NAME(config),{}},
        {EXOS_DATASET_BROWSE_NAME(config.maxSpeed),{}},
        {EXOS_DATASET_BROWSE_NAME(config.minSpeed),{}},
        {EXOS_DATASET_BROWSE_NAME(config.baseWidth),{}},
        {EXOS_DATASET_BROWSE_NAME(encoder),{}},
        {EXOS_DATASET_BROWSE_NAME(encoder.encoder1),{}},
        {EXOS_DATASET_BROWSE_NAME(encoder.encoder2),{}},
        {EXOS_DATASET_BROWSE_NAME(vaccumTopic),{}},
        {EXOS_DATASET_BROWSE_NAME(vaccumTopic.vaccumValve),{}},
        {EXOS_DATASET_BROWSE_NAME(vaccumTopic.vaccumMotor),{}},
        {EXOS_DATASET_BROWSE_NAME(lineFollow),{}},
        {EXOS_DATASET_BROWSE_NAME(lineFollow.lineMode),{}},
        {EXOS_DATASET_BROWSE_NAME(lineFollow.lineSharpTurn),{}},
        {EXOS_DATASET_BROWSE_NAME(lineFollow.lineHoldRight),{}},
        {EXOS_DATASET_BROWSE_NAME(lineFollow.lineForward),{}},
        {EXOS_DATASET_BROWSE_NAME(lineFollow.lineInterSection),{}},
        {EXOS_DATASET_BROWSE_NAME(lineFollow.lineDecision),{}},
        {EXOS_DATASET_BROWSE_NAME(lineFollow.lineFast),{}},
        {EXOS_DATASET_BROWSE_NAME(lineFollow.lineSlow),{}},
        {EXOS_DATASET_BROWSE_NAME(lineStatus),{}},
        {EXOS_DATASET_BROWSE_NAME(lineStatus.lineStatusCode),{}}
    };

    exos_datamodel_calc_dataset_info(datasets, sizeof(datasets));

    return exos_datamodel_connect(datamodel, config_ros_topics_typ, datasets, sizeof(datasets), datamodel_event_callback);
}
```
